Yaskawa INFORM job: miniTRJ0.JBI

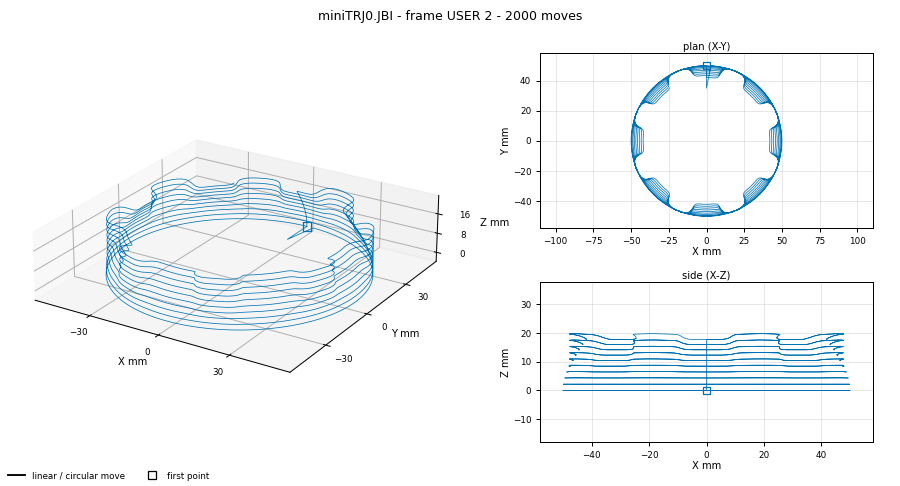
[picture p0: tool path of miniTRJ0.JBI in frame USER 2, 2000 of 2000 moves have a stored position in this frame; points joined in program order, loops and branches not executed]
/JOB
//NAME miniTRJ0
//POS
///NPOS 2000,0,0,0,0,0
///USER 2
///TOOL 1
///POSTYPE USER
///RECTAN
///RCONF 1,0,0,0,0,0,0,0,0,0,0,0,0,0,0,0,0,0,0,0,0,0,0,0
C00000=0.000,50.000,0.000,143.3809,0.0008,0.0000
C00001=0.000,35.000,0.000,143.3809,0.0008,0.0000
C00002=2.896,49.916,0.000,143.4142,-2.1763,0.0000
C00003=5.494,49.697,0.000,143.4861,-2.5054,0.0000
C00004=7.782,49.391,0.000,143.6143,-1.9514,0.0000
C00005=9.349,49.118,0.000,143.7421,-1.4817,0.0000
C00006=10.427,48.901,0.000,143.8463,-1.1243,0.0000
C00007=11.297,48.707,0.000,143.9396,-0.8206,0.0000
C00008=12.176,48.495,0.000,144.0418,-0.5020,0.0000
C00009=13.275,48.206,0.000,144.1803,-0.0901,0.0000
C00010=14.624,47.814,0.000,144.3651,0.4321,0.0000
C00011=16.047,47.355,0.000,144.5758,0.9982,0.0000
C00012=17.369,46.886,0.000,144.7843,1.5341,0.0000
C00013=18.561,46.427,0.000,144.9812,2.0219,0.0000
C00014=19.705,45.953,0.000,155.0622,-25.4971,0.0000
C00015=20.871,45.435,0.000,154.5493,-25.2482,0.0000
C00016=22.138,44.832,0.000,153.9948,-24.9681,0.0000
C00017=23.469,44.150,0.000,153.4198,-24.6638,0.0000
C00018=24.700,43.473,0.000,152.9002,-24.3753,0.0000
C00019=25.682,42.901,0.000,152.4981,-24.1419,0.0000
C00020=26.453,42.429,0.000,152.1923,-23.9575,0.0000
C00021=27.205,41.951,0.000,151.9052,-23.7787,0.0000
C00022=28.121,41.343,0.000,151.5731,-23.5641,0.0000
C00023=29.422,40.427,0.000,151.1462,-23.2751,0.0000
C00024=31.256,39.026,0.000,150.6643,-22.9190,0.0000
C00025=33.248,37.344,0.000,150.8238,-23.2222,0.0000
C00026=35.355,35.355,0.000,152.2782,-24.9479,0.0000
C00027=37.344,33.248,0.000,153.8299,-26.6153,0.0000
C00028=39.026,31.256,0.000,154.1264,-26.8237,0.0000
C00029=40.427,29.422,0.000,153.8428,-26.3144,0.0000
C00030=41.343,28.121,0.000,153.6210,-25.8703,0.0000
C00031=41.951,27.205,0.000,153.4595,-25.5278,0.0000
C00032=42.429,26.453,0.000,153.3270,-25.2337,0.0000
C00033=42.901,25.682,0.000,153.1924,-24.9221,0.0000
C00034=43.473,24.700,0.000,153.0248,-24.5152,0.0000
C00035=44.150,23.469,0.000,152.8218,-23.9932,0.0000
C00036=44.832,22.138,0.000,152.6122,-23.4205,0.0000
C00037=45.435,20.871,0.000,152.4232,-22.8724,0.0000
C00038=45.953,19.705,0.000,152.2582,-22.3690,0.0000
C00039=46.427,18.561,0.000,-177.5317,-34.9939,0.0000
C00040=46.886,17.369,0.000,-178.1225,-35.2012,0.0000
C00041=47.355,16.047,0.000,-178.7751,-35.4180,0.0000
C00042=47.814,14.624,0.000,-179.4684,-35.6337,0.0000
C00043=48.206,13.275,0.000,179.8889,-35.8197,0.0000
C00044=48.495,12.176,0.000,179.3798,-35.9566,0.0000
C00045=48.707,11.297,0.000,178.9849,-36.0561,0.0000
C00046=48.901,10.427,0.000,178.6076,-36.1456,0.0000
C00047=49.118,9.349,0.000,178.1627,-36.2439,0.0000
C00048=49.391,7.782,0.000,177.5765,-36.3612,0.0000
C00049=49.697,5.494,0.000,176.8838,-36.4734,0.0000
C00050=49.916,2.896,0.000,177.2904,-36.5551,0.0000
C00051=50.000,0.000,0.000,-179.9990,-36.6191,0.0000
C00052=49.916,-2.896,0.000,-177.2909,-36.5552,0.0000
C00053=49.697,-5.494,0.000,-176.8841,-36.4733,0.0000
C00054=49.391,-7.782,0.000,-177.5773,-36.3612,0.0000
C00055=49.118,-9.349,0.000,-178.1633,-36.2439,0.0000
C00056=48.901,-10.427,0.000,-178.6081,-36.1456,0.0000
C00057=48.707,-11.297,0.000,-178.9853,-36.0561,0.0000
C00058=48.495,-12.176,0.000,-179.3801,-35.9565,0.0000
C00059=48.206,-13.275,0.000,-179.8890,-35.8196,0.0000
C00060=47.814,-14.624,0.000,179.4684,-35.6336,0.0000
C00061=47.355,-16.047,0.000,178.7752,-35.4179,0.0000
C00062=46.886,-17.369,0.000,178.1227,-35.2010,0.0000
C00063=46.427,-18.561,0.000,177.5319,-34.9937,0.0000
C00064=45.953,-19.705,0.000,-152.2579,-22.3690,0.0000
C00065=45.435,-20.871,0.000,-152.4230,-22.8724,0.0000
C00066=44.832,-22.138,0.000,-152.6120,-23.4205,0.0000
C00067=44.150,-23.469,0.000,-152.8217,-23.9933,0.0000
C00068=43.473,-24.700,0.000,-153.0248,-24.5153,0.0000
C00069=42.901,-25.682,0.000,-153.1925,-24.9223,0.0000
C00070=42.429,-26.453,0.000,-153.3272,-25.2339,0.0000
C00071=41.951,-27.205,0.000,-153.4597,-25.5281,0.0000
C00072=41.343,-28.121,0.000,-153.6213,-25.8707,0.0000
C00073=40.427,-29.422,0.000,-153.8432,-26.3148,0.0000
C00074=39.026,-31.256,0.000,-154.1266,-26.8239,0.0000
C00075=37.344,-33.248,0.000,-153.8302,-26.6155,0.0000
C00076=35.355,-35.355,0.000,-152.2770,-24.9466,0.0000
C00077=33.248,-37.344,0.000,-150.8240,-23.2225,0.0000
C00078=31.256,-39.026,0.000,-150.6645,-22.9191,0.0000
C00079=29.422,-40.427,0.000,-151.1466,-23.2756,0.0000
C00080=28.121,-41.343,0.000,-151.5735,-23.5644,0.0000
C00081=27.205,-41.951,0.000,-151.9055,-23.7790,0.0000
C00082=26.453,-42.429,0.000,-152.1925,-23.9578,0.0000
C00083=25.682,-42.901,0.000,-152.4983,-24.1420,0.0000
C00084=24.700,-43.473,0.000,-152.9003,-24.3754,0.0000
C00085=23.469,-44.150,0.000,-153.4199,-24.6637,0.0000
C00086=22.138,-44.832,0.000,-153.9949,-24.9680,0.0000
C00087=20.871,-45.435,0.000,-154.5494,-25.2480,0.0000
C00088=19.705,-45.953,0.000,-155.0622,-25.4968,0.0000
C00089=18.561,-46.427,0.000,-144.9812,2.0219,0.0000
C00090=17.369,-46.886,0.000,-144.7843,1.5341,0.0000
C00091=16.047,-47.355,0.000,-144.5758,0.9982,0.0000
C00092=14.624,-47.814,0.000,-144.3651,0.4321,0.0000
C00093=13.275,-48.206,0.000,-144.1803,-0.0901,0.0000
C00094=12.176,-48.495,0.000,-144.0418,-0.5020,0.0000
C00095=11.297,-48.707,0.000,-143.9396,-0.8206,0.0000
C00096=10.427,-48.901,0.000,-143.8463,-1.1243,0.0000
C00097=9.349,-49.118,0.000,-143.7421,-1.4817,0.0000
C00098=7.782,-49.391,0.000,-143.6143,-1.9514,0.0000
C00099=5.494,-49.697,0.000,-143.4861,-2.5054,0.0000
C00100=2.896,-49.916,0.000,-143.4142,-2.1763,0.0000
C00101=0.000,-50.000,0.000,-143.3809,0.0008,0.0000
C00102=0.000,-50.000,0.000,-143.3809,0.0008,0.0000
C00103=-2.896,-49.916,0.000,-143.4141,2.1759,0.0000
C00104=-5.494,-49.697,0.000,-143.4861,2.5052,0.0000
C00105=-7.782,-49.391,0.000,-143.6143,1.9508,0.0000
C00106=-9.349,-49.118,0.000,-143.7421,1.4812,0.0000
C00107=-10.427,-48.901,0.000,-143.8463,1.1239,0.0000
C00108=-11.297,-48.707,0.000,-143.9396,0.8203,0.0000
C00109=-12.176,-48.495,0.000,-144.0419,0.5018,0.0000
C00110=-13.275,-48.206,0.000,-144.1804,0.0900,0.0000
C00111=-14.624,-47.814,0.000,-144.3652,-0.4320,0.0000
C00112=-16.047,-47.355,0.000,-144.5759,-0.9981,0.0000
C00113=-17.369,-46.886,0.000,-144.7845,-1.5339,0.0000
C00114=-18.561,-46.427,0.000,-144.9813,-2.0217,0.0000
C00115=-19.705,-45.953,0.000,-155.0622,25.4971,0.0000
C00116=-20.871,-45.435,0.000,-154.5493,25.2482,0.0000
C00117=-22.138,-44.832,0.000,-153.9948,24.9681,0.0000
C00118=-23.469,-44.150,0.000,-153.4198,24.6638,0.0000
C00119=-24.700,-43.473,0.000,-152.9002,24.3753,0.0000
C00120=-25.682,-42.901,0.000,-152.4981,24.1419,0.0000
C00121=-26.453,-42.429,0.000,-152.1923,23.9575,0.0000
C00122=-27.205,-41.951,0.000,-151.9052,23.7787,0.0000
C00123=-28.121,-41.343,0.000,-151.5731,23.5641,0.0000
C00124=-29.422,-40.427,0.000,-151.1462,23.2751,0.0000
C00125=-31.256,-39.026,0.000,-150.6643,22.9190,0.0000
C00126=-33.248,-37.344,0.000,-150.8238,23.2222,0.0000
C00127=-35.355,-35.355,0.000,-152.2782,24.9479,0.0000
C00128=-37.344,-33.248,0.000,-153.8299,26.6153,0.0000
C00129=-39.026,-31.256,0.000,-154.1264,26.8237,0.0000
C00130=-40.427,-29.422,0.000,-153.8428,26.3144,0.0000
C00131=-41.343,-28.121,0.000,-153.6210,25.8703,0.0000
C00132=-41.951,-27.205,0.000,-153.4595,25.5278,0.0000
C00133=-42.429,-26.453,0.000,-153.3270,25.2337,0.0000
C00134=-42.901,-25.682,0.000,-153.1924,24.9221,0.0000
C00135=-43.473,-24.700,0.000,-153.0248,24.5152,0.0000
C00136=-44.150,-23.469,0.000,-152.8218,23.9932,0.0000
C00137=-44.832,-22.138,0.000,-152.6122,23.4205,0.0000
C00138=-45.435,-20.871,0.000,-152.4232,22.8724,0.0000
C00139=-45.953,-19.705,0.000,-152.2582,22.3690,0.0000
C00140=-46.427,-18.561,0.000,177.5317,34.9939,0.0000
C00141=-46.886,-17.369,0.000,178.1225,35.2012,0.0000
C00142=-47.355,-16.047,0.000,178.7751,35.4180,0.0000
C00143=-47.814,-14.624,0.000,179.4684,35.6337,0.0000
C00144=-48.206,-13.275,0.000,-179.8889,35.8197,0.0000
C00145=-48.495,-12.176,0.000,-179.3798,35.9566,0.0000
C00146=-48.707,-11.297,0.000,-178.9849,36.0561,0.0000
C00147=-48.901,-10.427,0.000,-178.6076,36.1456,0.0000
C00148=-49.118,-9.349,0.000,-178.1627,36.2439,0.0000
C00149=-49.391,-7.782,0.000,-177.5765,36.3612,0.0000
C00150=-49.697,-5.494,0.000,-176.8838,36.4734,0.0000
C00151=-49.916,-2.896,0.000,-177.2904,36.5551,0.0000
C00152=-50.000,0.000,0.000,179.9990,36.6191,0.0000
C00153=-49.916,2.896,0.000,177.2909,36.5552,0.0000
C00154=-49.697,5.494,0.000,176.8841,36.4733,0.0000
C00155=-49.391,7.782,0.000,177.5773,36.3612,0.0000
C00156=-49.118,9.349,0.000,178.1633,36.2439,0.0000
C00157=-48.901,10.427,0.000,178.6081,36.1456,0.0000
C00158=-48.707,11.297,0.000,178.9853,36.0561,0.0000
C00159=-48.495,12.176,0.000,179.3801,35.9565,0.0000
C00160=-48.206,13.275,0.000,179.8890,35.8196,0.0000
C00161=-47.814,14.624,0.000,-179.4684,35.6336,0.0000
C00162=-47.355,16.047,0.000,-178.7752,35.4179,0.0000
C00163=-46.886,17.369,0.000,-178.1227,35.2010,0.0000
C00164=-46.427,18.561,0.000,-177.5319,34.9937,0.0000
C00165=-45.953,19.705,0.000,152.2579,22.3690,0.0000
C00166=-45.435,20.871,0.000,152.4230,22.8724,0.0000
C00167=-44.832,22.138,0.000,152.6120,23.4205,0.0000
C00168=-44.150,23.469,0.000,152.8217,23.9933,0.0000
C00169=-43.473,24.700,0.000,153.0248,24.5153,0.0000
C00170=-42.901,25.682,0.000,153.1925,24.9223,0.0000
C00171=-42.429,26.453,0.000,153.3272,25.2339,0.0000
C00172=-41.951,27.205,0.000,153.4597,25.5281,0.0000
C00173=-41.343,28.121,0.000,153.6213,25.8707,0.0000
C00174=-40.427,29.422,0.000,153.8432,26.3148,0.0000
C00175=-39.026,31.256,0.000,154.1266,26.8239,0.0000
C00176=-37.344,33.248,0.000,153.8302,26.6155,0.0000
C00177=-35.355,35.355,0.000,152.2770,24.9466,0.0000
C00178=-33.248,37.344,0.000,150.8240,23.2225,0.0000
C00179=-31.256,39.026,0.000,150.6645,22.9191,0.0000
C00180=-29.422,40.427,0.000,151.1466,23.2756,0.0000
C00181=-28.121,41.343,0.000,151.5735,23.5644,0.0000
C00182=-27.205,41.951,0.000,151.9055,23.7790,0.0000
C00183=-26.453,42.429,0.000,152.1925,23.9578,0.0000
C00184=-25.682,42.901,0.000,152.4983,24.1420,0.0000
C00185=-24.700,43.473,0.000,152.9003,24.3754,0.0000
C00186=-23.469,44.150,0.000,153.4199,24.6637,0.0000
C00187=-22.138,44.832,0.000,153.9949,24.9680,0.0000
C00188=-20.871,45.435,0.000,154.5494,25.2480,0.0000
C00189=-19.705,45.953,0.000,155.0622,25.4968,0.0000
C00190=-18.561,46.427,0.000,144.9813,-2.0217,0.0000
C00191=-17.369,46.886,0.000,144.7845,-1.5339,0.0000
C00192=-16.047,47.355,0.000,144.5759,-0.9981,0.0000
C00193=-14.624,47.814,0.000,144.3652,-0.4320,0.0000
C00194=-13.275,48.206,0.000,144.1804,0.0900,0.0000
C00195=-12.176,48.495,0.000,144.0419,0.5018,0.0000
C00196=-11.297,48.707,0.000,143.9396,0.8203,0.0000
C00197=-10.427,48.901,0.000,143.8463,1.1239,0.0000
C00198=-9.349,49.118,0.000,143.7421,1.4812,0.0000
C00199=-7.782,49.391,0.000,143.6143,1.9508,0.0000
C00200=-5.494,49.697,0.000,143.4861,2.5052,0.0000
C00201=-2.896,49.916,0.000,143.4141,2.1759,0.0000
C00202=0.000,50.000,0.000,143.3809,0.0008,0.0000
C00203=0.000,49.846,2.195,142.7871,0.0008,0.0000
C00204=2.882,49.762,2.195,142.8227,-2.2150,0.0000
C00205=5.471,49.545,2.195,142.8908,-2.4632,0.0000
C00206=7.753,49.245,2.195,143.0117,-1.8435,0.0000
C00207=9.315,48.989,2.196,143.1359,-1.3366,0.0000
C00208=10.389,48.795,2.197,143.2401,-0.9560,0.0000
C00209=11.257,48.629,2.198,143.3352,-0.6346,0.0000
C00210=12.134,48.445,2.199,143.4401,-0.2988,0.0000
C00211=13.230,48.181,2.199,143.5809,0.1341,0.0000
C00212=14.582,47.809,2.200,143.7697,0.6839,0.0000
C00213=16.014,47.361,2.200,143.9865,1.2808,0.0000
C00214=17.348,46.893,2.200,144.2028,1.8461,0.0000
C00215=18.554,46.430,2.200,144.4088,2.3605,0.0000
C00216=19.712,45.950,2.200,154.8156,-26.1236,0.0000
C00217=20.891,45.426,2.200,154.2738,-25.8594,0.0000
C00218=22.166,44.813,2.200,153.6898,-25.5604,0.0000
C00219=23.495,44.117,2.200,153.0860,-25.2351,0.0000
C00220=24.714,43.424,2.199,152.5422,-24.9264,0.0000
C00221=25.676,42.836,2.199,152.1226,-24.6771,0.0000
C00222=26.426,42.346,2.198,151.8021,-24.4802,0.0000
C00223=27.157,41.850,2.197,151.5007,-24.2879,0.0000
C00224=28.054,41.227,2.196,151.1523,-24.0540,0.0000
C00225=29.339,40.304,2.195,150.7028,-23.7323,0.0000
C00226=31.165,38.902,2.195,150.1829,-23.3183,0.0000
C00227=33.149,37.225,2.195,150.2905,-23.5560,0.0000
C00228=35.246,35.246,2.195,151.7659,-25.3187,0.0000
C00229=37.225,33.149,2.195,153.3450,-27.0199,0.0000
C00230=38.902,31.165,2.195,153.5809,-27.1689,0.0000
C00231=40.304,29.339,2.195,153.2459,-26.6124,0.0000
C00232=41.227,28.054,2.196,152.9964,-26.1408,0.0000
C00233=41.850,27.157,2.197,152.8199,-25.7796,0.0000
C00234=42.346,26.426,2.198,152.6780,-25.4699,0.0000
C00235=42.836,25.676,2.199,152.5351,-25.1428,0.0000
C00236=43.424,24.714,2.199,152.3569,-24.7173,0.0000
C00237=44.117,23.495,2.200,152.1408,-24.1705,0.0000
C00238=44.813,22.166,2.200,151.9184,-23.5689,0.0000
C00239=45.426,20.891,2.200,151.7187,-22.9922,0.0000
C00240=45.950,19.712,2.200,151.5461,-22.4615,0.0000
C00241=46.430,18.554,2.200,-177.0981,-35.5564,0.0000
C00242=46.893,17.348,2.200,-177.7244,-35.7758,0.0000
C00243=47.361,16.014,2.200,-178.4168,-36.0031,0.0000
C00244=47.809,14.582,2.200,-179.1522,-36.2274,0.0000
C00245=48.181,13.230,2.199,-179.8333,-36.4190,0.0000
C00246=48.445,12.134,2.199,179.6280,-36.5594,0.0000
C00247=48.629,11.257,2.198,179.2089,-36.6622,0.0000
C00248=48.795,10.389,2.197,178.8068,-36.7540,0.0000
C00249=48.989,9.315,2.196,178.3295,-36.8524,0.0000
C00250=49.245,7.753,2.195,177.6925,-36.9660,0.0000
C00251=49.545,5.471,2.195,176.9123,-37.0692,0.0000
C00252=49.762,2.882,2.195,177.2208,-37.1449,0.0000
C00253=49.846,0.000,2.195,-179.9990,-37.2129,0.0000
C00254=49.762,-2.882,2.195,-177.2212,-37.1450,0.0000
C00255=49.545,-5.471,2.195,-176.9127,-37.0691,0.0000
C00256=49.245,-7.753,2.195,-177.6932,-36.9659,0.0000
C00257=48.989,-9.315,2.196,-178.3302,-36.8524,0.0000
C00258=48.795,-10.389,2.197,-178.8073,-36.7540,0.0000
C00259=48.629,-11.257,2.198,-179.2093,-36.6621,0.0000
C00260=48.445,-12.134,2.199,-179.6283,-36.5593,0.0000
C00261=48.181,-13.230,2.199,179.8332,-36.4189,0.0000
C00262=47.809,-14.582,2.200,179.1522,-36.2273,0.0000
C00263=47.361,-16.014,2.200,178.4168,-36.0030,0.0000
C00264=46.893,-17.348,2.200,177.7245,-35.7757,0.0000
C00265=46.430,-18.554,2.200,177.0983,-35.5563,0.0000
C00266=45.950,-19.712,2.200,-151.5459,-22.4615,0.0000
C00267=45.426,-20.891,2.200,-151.7185,-22.9922,0.0000
C00268=44.813,-22.166,2.200,-151.9182,-23.5690,0.0000
C00269=44.117,-23.495,2.200,-152.1407,-24.1705,0.0000
C00270=43.424,-24.714,2.199,-152.3570,-24.7174,0.0000
C00271=42.836,-25.676,2.199,-152.5352,-25.1430,0.0000
C00272=42.346,-26.426,2.198,-152.6781,-25.4702,0.0000
C00273=41.850,-27.157,2.197,-152.8202,-25.7800,0.0000
C00274=41.227,-28.054,2.196,-152.9968,-26.1412,0.0000
C00275=40.304,-29.339,2.195,-153.2463,-26.6128,0.0000
C00276=38.902,-31.165,2.195,-153.5811,-27.1692,0.0000
C00277=37.225,-33.149,2.195,-153.3453,-27.0201,0.0000
C00278=35.246,-35.246,2.195,-151.7648,-25.3174,0.0000
C00279=33.149,-37.225,2.195,-150.2907,-23.5563,0.0000
C00280=31.165,-38.902,2.195,-150.1831,-23.3185,0.0000
C00281=29.339,-40.304,2.195,-150.7032,-23.7328,0.0000
C00282=28.054,-41.227,2.196,-151.1526,-24.0544,0.0000
C00283=27.157,-41.850,2.197,-151.5010,-24.2882,0.0000
C00284=26.426,-42.346,2.198,-151.8023,-24.4804,0.0000
C00285=25.676,-42.836,2.199,-152.1228,-24.6773,0.0000
C00286=24.714,-43.424,2.199,-152.5424,-24.9265,0.0000
C00287=23.495,-44.117,2.200,-153.0861,-25.2350,0.0000
C00288=22.166,-44.813,2.200,-153.6898,-25.5603,0.0000
C00289=20.891,-45.426,2.200,-154.2738,-25.8592,0.0000
C00290=19.712,-45.950,2.200,-154.8157,-26.1234,0.0000
C00291=18.554,-46.430,2.200,-144.4088,2.3605,0.0000
C00292=17.348,-46.893,2.200,-144.2028,1.8461,0.0000
C00293=16.014,-47.361,2.200,-143.9865,1.2808,0.0000
C00294=14.582,-47.809,2.200,-143.7697,0.6839,0.0000
C00295=13.230,-48.181,2.199,-143.5809,0.1341,0.0000
C00296=12.134,-48.445,2.199,-143.4401,-0.2988,0.0000
C00297=11.257,-48.629,2.198,-143.3352,-0.6346,0.0000
C00298=10.389,-48.795,2.197,-143.2401,-0.9560,0.0000
C00299=9.315,-48.989,2.196,-143.1359,-1.3366,0.0000
C00300=7.753,-49.245,2.195,-143.0117,-1.8435,0.0000
C00301=5.471,-49.545,2.195,-142.8908,-2.4632,0.0000
C00302=2.882,-49.762,2.195,-142.8227,-2.2150,0.0000
C00303=0.000,-49.846,2.195,-142.7871,0.0008,0.0000
C00304=0.000,-49.846,2.195,-142.7871,0.0008,0.0000
C00305=-2.882,-49.762,2.195,-142.8226,2.2147,0.0000
C00306=-5.471,-49.545,2.195,-142.8908,2.4630,0.0000
C00307=-7.753,-49.245,2.195,-143.0117,1.8429,0.0000
C00308=-9.315,-48.989,2.196,-143.1359,1.3361,0.0000
C00309=-10.389,-48.795,2.197,-143.2401,0.9556,0.0000
C00310=-11.257,-48.629,2.198,-143.3353,0.6342,0.0000
C00311=-12.134,-48.445,2.199,-143.4401,0.2985,0.0000
C00312=-13.230,-48.181,2.199,-143.5810,-0.1342,0.0000
C00313=-14.582,-47.809,2.200,-143.7698,-0.6839,0.0000
C00314=-16.014,-47.361,2.200,-143.9866,-1.2807,0.0000
C00315=-17.348,-46.893,2.200,-144.2029,-1.8459,0.0000
C00316=-18.554,-46.430,2.200,-144.4089,-2.3603,0.0000
C00317=-19.712,-45.950,2.200,-154.8156,26.1236,0.0000
C00318=-20.891,-45.426,2.200,-154.2738,25.8594,0.0000
C00319=-22.166,-44.813,2.200,-153.6898,25.5604,0.0000
C00320=-23.495,-44.117,2.200,-153.0860,25.2351,0.0000
C00321=-24.714,-43.424,2.199,-152.5422,24.9264,0.0000
C00322=-25.676,-42.836,2.199,-152.1226,24.6771,0.0000
C00323=-26.426,-42.346,2.198,-151.8021,24.4802,0.0000
C00324=-27.157,-41.850,2.197,-151.5007,24.2879,0.0000
C00325=-28.054,-41.227,2.196,-151.1523,24.0540,0.0000
C00326=-29.339,-40.304,2.195,-150.7028,23.7323,0.0000
C00327=-31.165,-38.902,2.195,-150.1829,23.3183,0.0000
C00328=-33.149,-37.225,2.195,-150.2905,23.5560,0.0000
C00329=-35.246,-35.246,2.195,-151.7659,25.3187,0.0000
C00330=-37.225,-33.149,2.195,-153.3450,27.0199,0.0000
C00331=-38.902,-31.165,2.195,-153.5809,27.1689,0.0000
C00332=-40.304,-29.339,2.195,-153.2459,26.6124,0.0000
C00333=-41.227,-28.054,2.196,-152.9964,26.1408,0.0000
C00334=-41.850,-27.157,2.197,-152.8199,25.7796,0.0000
C00335=-42.346,-26.426,2.198,-152.6780,25.4699,0.0000
C00336=-42.836,-25.676,2.199,-152.5351,25.1428,0.0000
C00337=-43.424,-24.714,2.199,-152.3569,24.7173,0.0000
C00338=-44.117,-23.495,2.200,-152.1408,24.1705,0.0000
C00339=-44.813,-22.166,2.200,-151.9184,23.5689,0.0000
C00340=-45.426,-20.891,2.200,-151.7187,22.9922,0.0000
C00341=-45.950,-19.712,2.200,-151.5461,22.4615,0.0000
C00342=-46.430,-18.554,2.200,177.0981,35.5564,0.0000
C00343=-46.893,-17.348,2.200,177.7244,35.7758,0.0000
C00344=-47.361,-16.014,2.200,178.4168,36.0031,0.0000
C00345=-47.809,-14.582,2.200,179.1522,36.2274,0.0000
C00346=-48.181,-13.230,2.199,179.8333,36.4190,0.0000
C00347=-48.445,-12.134,2.199,-179.6280,36.5594,0.0000
C00348=-48.629,-11.257,2.198,-179.2089,36.6622,0.0000
C00349=-48.795,-10.389,2.197,-178.8068,36.7540,0.0000
C00350=-48.989,-9.315,2.196,-178.3295,36.8524,0.0000
C00351=-49.245,-7.753,2.195,-177.6925,36.9660,0.0000
C00352=-49.545,-5.471,2.195,-176.9123,37.0692,0.0000
C00353=-49.762,-2.882,2.195,-177.2208,37.1449,0.0000
C00354=-49.846,0.000,2.195,179.9990,37.2129,0.0000
C00355=-49.762,2.882,2.195,177.2212,37.1450,0.0000
C00356=-49.545,5.471,2.195,176.9127,37.0691,0.0000
C00357=-49.245,7.753,2.195,177.6932,36.9659,0.0000
C00358=-48.989,9.315,2.196,178.3302,36.8524,0.0000
C00359=-48.795,10.389,2.197,178.8073,36.7540,0.0000
C00360=-48.629,11.257,2.198,179.2093,36.6621,0.0000
C00361=-48.445,12.134,2.199,179.6283,36.5593,0.0000
C00362=-48.181,13.230,2.199,-179.8332,36.4189,0.0000
C00363=-47.809,14.582,2.200,-179.1522,36.2273,0.0000
C00364=-47.361,16.014,2.200,-178.4168,36.0030,0.0000
C00365=-46.893,17.348,2.200,-177.7245,35.7757,0.0000
C00366=-46.430,18.554,2.200,-177.0983,35.5563,0.0000
C00367=-45.950,19.712,2.200,151.5459,22.4615,0.0000
C00368=-45.426,20.891,2.200,151.7185,22.9922,0.0000
C00369=-44.813,22.166,2.200,151.9182,23.5690,0.0000
C00370=-44.117,23.495,2.200,152.1407,24.1705,0.0000
C00371=-43.424,24.714,2.199,152.3570,24.7174,0.0000
C00372=-42.836,25.676,2.199,152.5352,25.1430,0.0000
C00373=-42.346,26.426,2.198,152.6781,25.4702,0.0000
C00374=-41.850,27.157,2.197,152.8202,25.7800,0.0000
C00375=-41.227,28.054,2.196,152.9968,26.1412,0.0000
C00376=-40.304,29.339,2.195,153.2463,26.6128,0.0000
C00377=-38.902,31.165,2.195,153.5811,27.1692,0.0000
C00378=-37.225,33.149,2.195,153.3453,27.0201,0.0000
C00379=-35.246,35.246,2.195,151.7648,25.3174,0.0000
C00380=-33.149,37.225,2.195,150.2907,23.5563,0.0000
C00381=-31.165,38.902,2.195,150.1831,23.3185,0.0000
C00382=-29.339,40.304,2.195,150.7032,23.7328,0.0000
C00383=-28.054,41.227,2.196,151.1526,24.0544,0.0000
C00384=-27.157,41.850,2.197,151.5010,24.2882,0.0000
C00385=-26.426,42.346,2.198,151.8023,24.4804,0.0000
C00386=-25.676,42.836,2.199,152.1228,24.6773,0.0000
C00387=-24.714,43.424,2.199,152.5424,24.9265,0.0000
C00388=-23.495,44.117,2.200,153.0861,25.2350,0.0000
C00389=-22.166,44.813,2.200,153.6898,25.5603,0.0000
C00390=-20.891,45.426,2.200,154.2738,25.8592,0.0000
C00391=-19.712,45.950,2.200,154.8157,26.1234,0.0000
C00392=-18.554,46.430,2.200,144.4089,-2.3603,0.0000
C00393=-17.348,46.893,2.200,144.2029,-1.8459,0.0000
C00394=-16.014,47.361,2.200,143.9866,-1.2807,0.0000
C00395=-14.582,47.809,2.200,143.7698,-0.6839,0.0000
C00396=-13.230,48.181,2.199,143.5810,-0.1342,0.0000
C00397=-12.134,48.445,2.199,143.4401,0.2985,0.0000
C00398=-11.257,48.629,2.198,143.3353,0.6342,0.0000
C00399=-10.389,48.795,2.197,143.2401,0.9556,0.0000
C00400=-9.315,48.989,2.196,143.1359,1.3361,0.0000
C00401=-7.753,49.245,2.195,143.0117,1.8429,0.0000
C00402=-5.471,49.545,2.195,142.8908,2.4630,0.0000
C00403=-2.882,49.762,2.195,142.8226,2.2147,0.0000
C00404=0.000,49.846,2.195,142.7871,0.0008,0.0000
C00405=0.000,49.410,4.351,142.2720,0.0007,0.0000
C00406=2.842,49.327,4.351,142.3092,-2.2444,0.0000
C00407=5.404,49.114,4.351,142.3736,-2.4180,0.0000
C00408=7.672,48.833,4.355,142.4892,-1.7397,0.0000
C00409=9.218,48.623,4.363,142.6124,-1.2036,0.0000
C00410=10.282,48.495,4.374,142.7197,-0.8069,0.0000
C00411=11.143,48.407,4.384,142.8211,-0.4739,0.0000
C00412=12.014,48.303,4.391,142.9335,-0.1276,0.0000
C00413=13.101,48.111,4.395,143.0816,0.3184,0.0000
C00414=14.461,47.794,4.396,143.2802,0.8931,0.0000
C00415=15.918,47.378,4.398,143.5102,1.5238,0.0000
C00416=17.289,46.913,4.399,143.7405,2.1264,0.0000
C00417=18.533,46.438,4.400,143.9621,2.6774,0.0000
C00418=19.732,45.942,4.400,154.6593,-26.6527,0.0000
C00419=20.948,45.397,4.399,154.0760,-26.3698,0.0000
C00420=22.246,44.758,4.398,153.4514,-26.0501,0.0000
C00421=23.570,44.021,4.396,152.8110,-25.7058,0.0000
C00422=24.756,43.284,4.395,152.2399,-25.3828,0.0000
C00423=25.660,42.651,4.391,151.8041,-25.1271,0.0000
C00424=26.350,42.108,4.384,151.4691,-24.9258,0.0000
C00425=27.021,41.562,4.374,151.1539,-24.7276,0.0000
C00426=27.864,40.900,4.363,150.7913,-24.4822,0.0000
C00427=29.106,39.955,4.355,150.3226,-24.1357,0.0000
C00428=30.908,38.550,4.351,149.7679,-23.6707,0.0000
C00429=32.870,36.889,4.351,149.8283,-23.8474,0.0000
C00430=34.938,34.938,4.351,151.3189,-25.6389,0.0000
C00431=36.889,32.870,4.351,152.9185,-27.3666,0.0000
C00432=38.550,30.908,4.351,153.0982,-27.4607,0.0000
C00433=39.955,29.106,4.355,152.7186,-26.8609,0.0000
C00434=40.900,27.864,4.363,152.4494,-26.3664,0.0000
C00435=41.562,27.021,4.374,152.2657,-25.9900,0.0000
C00436=42.108,26.350,4.384,152.1223,-25.6669,0.0000
C00437=42.651,25.660,4.391,151.9798,-25.3262,0.0000
C00438=43.284,24.756,4.395,151.8006,-24.8854,0.0000
C00439=44.021,23.570,4.396,151.5781,-24.3120,0.0000
C00440=44.758,22.246,4.398,151.3465,-23.6751,0.0000
C00441=45.397,20.948,4.399,151.1361,-23.0596,0.0000
C00442=45.942,19.732,4.400,150.9546,-22.4900,0.0000
C00443=46.438,18.533,4.400,-176.6903,-35.9924,0.0000
C00444=46.913,17.289,4.399,-177.3636,-36.2306,0.0000
C00445=47.378,15.918,4.398,-178.1049,-36.4748,0.0000
C00446=47.794,14.461,4.396,-178.8858,-36.7146,0.0000
C00447=48.111,13.101,4.395,-179.6018,-36.9177,0.0000
C00448=48.303,12.014,4.391,179.8401,-37.0664,0.0000
C00449=48.407,11.143,4.384,179.4052,-37.1774,0.0000
C00450=48.495,10.282,4.374,178.9860,-37.2759,0.0000
C00451=48.623,9.218,4.363,178.4853,-37.3780,0.0000
C00452=48.833,7.672,4.355,177.8073,-37.4905,0.0000
C00453=49.114,5.404,4.351,176.9481,-37.5871,0.0000
C00454=49.327,2.842,4.351,177.1646,-37.6569,0.0000
C00455=49.410,0.000,4.351,-179.9991,-37.7280,0.0000
C00456=49.327,-2.842,4.351,-177.1650,-37.6569,0.0000
C00457=49.114,-5.404,4.351,-176.9485,-37.5870,0.0000
C00458=48.833,-7.672,4.355,-177.8080,-37.4905,0.0000
C00459=48.623,-9.218,4.363,-178.4859,-37.3779,0.0000
C00460=48.495,-10.282,4.374,-178.9865,-37.2759,0.0000
C00461=48.407,-11.143,4.384,-179.4056,-37.1773,0.0000
C00462=48.303,-12.014,4.391,-179.8405,-37.0663,0.0000
C00463=48.111,-13.101,4.395,179.6016,-36.9176,0.0000
C00464=47.794,-14.461,4.396,178.8858,-36.7145,0.0000
C00465=47.378,-15.918,4.398,178.1050,-36.4747,0.0000
C00466=46.913,-17.289,4.399,177.3637,-36.2305,0.0000
C00467=46.438,-18.533,4.400,176.6904,-35.9923,0.0000
C00468=45.942,-19.732,4.400,-150.9544,-22.4899,0.0000
C00469=45.397,-20.948,4.399,-151.1359,-23.0596,0.0000
C00470=44.758,-22.246,4.398,-151.3464,-23.6751,0.0000
C00471=44.021,-23.570,4.396,-151.5781,-24.3121,0.0000
C00472=43.284,-24.756,4.395,-151.8007,-24.8855,0.0000
C00473=42.651,-25.660,4.391,-151.9800,-25.3265,0.0000
C00474=42.108,-26.350,4.384,-152.1225,-25.6672,0.0000
C00475=41.562,-27.021,4.374,-152.2659,-25.9903,0.0000
C00476=40.900,-27.864,4.363,-152.4497,-26.3668,0.0000
C00477=39.955,-29.106,4.355,-152.7190,-26.8614,0.0000
C00478=38.550,-30.908,4.351,-153.0984,-27.4609,0.0000
C00479=36.889,-32.870,4.351,-152.9188,-27.3668,0.0000
C00480=34.938,-34.938,4.351,-151.3179,-25.6377,0.0000
C00481=32.870,-36.889,4.351,-149.8284,-23.8476,0.0000
C00482=30.908,-38.550,4.351,-149.7681,-23.6709,0.0000
C00483=29.106,-39.955,4.355,-150.3230,-24.1362,0.0000
C00484=27.864,-40.900,4.363,-150.7917,-24.4825,0.0000
C00485=27.021,-41.562,4.374,-151.1543,-24.7279,0.0000
C00486=26.350,-42.108,4.384,-151.4694,-24.9261,0.0000
C00487=25.660,-42.651,4.391,-151.8043,-25.1272,0.0000
C00488=24.756,-43.284,4.395,-152.2401,-25.3829,0.0000
C00489=23.570,-44.021,4.396,-152.8111,-25.7058,0.0000
C00490=22.246,-44.758,4.398,-153.4515,-26.0500,0.0000
C00491=20.948,-45.397,4.399,-154.0760,-26.3696,0.0000
C00492=19.732,-45.942,4.400,-154.6593,-26.6525,0.0000
C00493=18.533,-46.438,4.400,-143.9621,2.6774,0.0000
C00494=17.289,-46.913,4.399,-143.7405,2.1264,0.0000
C00495=15.918,-47.378,4.398,-143.5102,1.5238,0.0000
C00496=14.461,-47.794,4.396,-143.2802,0.8931,0.0000
C00497=13.101,-48.111,4.395,-143.0816,0.3184,0.0000
C00498=12.014,-48.303,4.391,-142.9335,-0.1276,0.0000
C00499=11.143,-48.407,4.384,-142.8211,-0.4739,0.0000
C00500=10.282,-48.495,4.374,-142.7197,-0.8069,0.0000
C00501=9.218,-48.623,4.363,-142.6124,-1.2036,0.0000
C00502=7.672,-48.833,4.355,-142.4892,-1.7397,0.0000
C00503=5.404,-49.114,4.351,-142.3736,-2.4180,0.0000
C00504=2.842,-49.327,4.351,-142.3092,-2.2444,0.0000
C00505=0.000,-49.410,4.351,-142.2720,0.0007,0.0000
C00506=0.000,-49.410,4.351,-142.2720,0.0007,0.0000
C00507=-2.842,-49.327,4.351,-142.3091,2.2441,0.0000
C00508=-5.404,-49.114,4.351,-142.3737,2.4177,0.0000
C00509=-7.672,-48.833,4.355,-142.4893,1.7391,0.0000
C00510=-9.218,-48.623,4.363,-142.6124,1.2031,0.0000
C00511=-10.282,-48.495,4.374,-142.7198,0.8065,0.0000
C00512=-11.143,-48.407,4.384,-142.8212,0.4736,0.0000
C00513=-12.014,-48.303,4.391,-142.9336,0.1273,0.0000
C00514=-13.101,-48.111,4.395,-143.0817,-0.3185,0.0000
C00515=-14.461,-47.794,4.396,-143.2803,-0.8932,0.0000
C00516=-15.918,-47.378,4.398,-143.5103,-1.5237,0.0000
C00517=-17.289,-46.913,4.399,-143.7406,-2.1263,0.0000
C00518=-18.533,-46.438,4.400,-143.9622,-2.6772,0.0000
C00519=-19.732,-45.942,4.400,-154.6593,26.6527,0.0000
C00520=-20.948,-45.397,4.399,-154.0760,26.3698,0.0000
C00521=-22.246,-44.758,4.398,-153.4514,26.0501,0.0000
C00522=-23.570,-44.021,4.396,-152.8110,25.7058,0.0000
C00523=-24.756,-43.284,4.395,-152.2399,25.3828,0.0000
C00524=-25.660,-42.651,4.391,-151.8041,25.1271,0.0000
C00525=-26.350,-42.108,4.384,-151.4691,24.9258,0.0000
C00526=-27.021,-41.562,4.374,-151.1539,24.7276,0.0000
C00527=-27.864,-40.900,4.363,-150.7913,24.4822,0.0000
C00528=-29.106,-39.955,4.355,-150.3226,24.1357,0.0000
C00529=-30.908,-38.550,4.351,-149.7679,23.6707,0.0000
C00530=-32.870,-36.889,4.351,-149.8283,23.8474,0.0000
C00531=-34.938,-34.938,4.351,-151.3189,25.6389,0.0000
C00532=-36.889,-32.870,4.351,-152.9185,27.3666,0.0000
C00533=-38.550,-30.908,4.351,-153.0982,27.4607,0.0000
C00534=-39.955,-29.106,4.355,-152.7186,26.8609,0.0000
C00535=-40.900,-27.864,4.363,-152.4494,26.3664,0.0000
C00536=-41.562,-27.021,4.374,-152.2657,25.9900,0.0000
C00537=-42.108,-26.350,4.384,-152.1223,25.6669,0.0000
C00538=-42.651,-25.660,4.391,-151.9798,25.3262,0.0000
C00539=-43.284,-24.756,4.395,-151.8006,24.8854,0.0000
C00540=-44.021,-23.570,4.396,-151.5781,24.3120,0.0000
C00541=-44.758,-22.246,4.398,-151.3465,23.6751,0.0000
C00542=-45.397,-20.948,4.399,-151.1361,23.0596,0.0000
C00543=-45.942,-19.732,4.400,-150.9546,22.4900,0.0000
C00544=-46.438,-18.533,4.400,176.6903,35.9924,0.0000
C00545=-46.913,-17.289,4.399,177.3636,36.2306,0.0000
C00546=-47.378,-15.918,4.398,178.1049,36.4748,0.0000
C00547=-47.794,-14.461,4.396,178.8858,36.7146,0.0000
C00548=-48.111,-13.101,4.395,179.6018,36.9177,0.0000
C00549=-48.303,-12.014,4.391,-179.8401,37.0664,0.0000
C00550=-48.407,-11.143,4.384,-179.4052,37.1774,0.0000
C00551=-48.495,-10.282,4.374,-178.9860,37.2759,0.0000
C00552=-48.623,-9.218,4.363,-178.4853,37.3780,0.0000
C00553=-48.833,-7.672,4.355,-177.8073,37.4905,0.0000
C00554=-49.114,-5.404,4.351,-176.9481,37.5871,0.0000
C00555=-49.327,-2.842,4.351,-177.1646,37.6569,0.0000
C00556=-49.410,0.000,4.351,179.9991,37.7280,0.0000
C00557=-49.327,2.842,4.351,177.1650,37.6569,0.0000
C00558=-49.114,5.404,4.351,176.9485,37.5870,0.0000
C00559=-48.833,7.672,4.355,177.8080,37.4905,0.0000
C00560=-48.623,9.218,4.363,178.4859,37.3779,0.0000
C00561=-48.495,10.282,4.374,178.9865,37.2759,0.0000
C00562=-48.407,11.143,4.384,179.4056,37.1773,0.0000
C00563=-48.303,12.014,4.391,179.8405,37.0663,0.0000
C00564=-48.111,13.101,4.395,-179.6016,36.9176,0.0000
C00565=-47.794,14.461,4.396,-178.8858,36.7145,0.0000
C00566=-47.378,15.918,4.398,-178.1050,36.4747,0.0000
C00567=-46.913,17.289,4.399,-177.3637,36.2305,0.0000
C00568=-46.438,18.533,4.400,-176.6904,35.9923,0.0000
C00569=-45.942,19.732,4.400,150.9544,22.4899,0.0000
C00570=-45.397,20.948,4.399,151.1359,23.0596,0.0000
C00571=-44.758,22.246,4.398,151.3464,23.6751,0.0000
C00572=-44.021,23.570,4.396,151.5781,24.3121,0.0000
C00573=-43.284,24.756,4.395,151.8007,24.8855,0.0000
C00574=-42.651,25.660,4.391,151.9800,25.3265,0.0000
C00575=-42.108,26.350,4.384,152.1225,25.6672,0.0000
C00576=-41.562,27.021,4.374,152.2659,25.9903,0.0000
C00577=-40.900,27.864,4.363,152.4497,26.3668,0.0000
C00578=-39.955,29.106,4.355,152.7190,26.8614,0.0000
C00579=-38.550,30.908,4.351,153.0984,27.4609,0.0000
C00580=-36.889,32.870,4.351,152.9188,27.3668,0.0000
C00581=-34.938,34.938,4.351,151.3179,25.6377,0.0000
C00582=-32.870,36.889,4.351,149.8284,23.8476,0.0000
C00583=-30.908,38.550,4.351,149.7681,23.6709,0.0000
C00584=-29.106,39.955,4.355,150.3230,24.1362,0.0000
C00585=-27.864,40.900,4.363,150.7917,24.4825,0.0000
C00586=-27.021,41.562,4.374,151.1543,24.7279,0.0000
C00587=-26.350,42.108,4.384,151.4694,24.9261,0.0000
C00588=-25.660,42.651,4.391,151.8043,25.1272,0.0000
C00589=-24.756,43.284,4.395,152.2401,25.3829,0.0000
C00590=-23.570,44.021,4.396,152.8111,25.7058,0.0000
C00591=-22.246,44.758,4.398,153.4515,26.0500,0.0000
C00592=-20.948,45.397,4.399,154.0760,26.3696,0.0000
C00593=-19.732,45.942,4.400,154.6593,26.6525,0.0000
C00594=-18.533,46.438,4.400,143.9622,-2.6772,0.0000
C00595=-17.289,46.913,4.399,143.7406,-2.1263,0.0000
C00596=-15.918,47.378,4.398,143.5103,-1.5237,0.0000
C00597=-14.461,47.794,4.396,143.2803,-0.8932,0.0000
C00598=-13.101,48.111,4.395,143.0817,-0.3185,0.0000
C00599=-12.014,48.303,4.391,142.9336,0.1273,0.0000
C00600=-11.143,48.407,4.384,142.8212,0.4736,0.0000
C00601=-10.282,48.495,4.374,142.7198,0.8065,0.0000
C00602=-9.218,48.623,4.363,142.6124,1.2031,0.0000
C00603=-7.672,48.833,4.355,142.4893,1.7391,0.0000
C00604=-5.404,49.114,4.351,142.3737,2.4177,0.0000
C00605=-2.842,49.327,4.351,142.3091,2.2441,0.0000
C00606=0.000,49.410,4.351,142.2720,0.0007,0.0000
C00607=0.000,48.740,6.447,141.8391,0.0007,0.0000
C00608=2.781,48.660,6.446,141.8776,-2.2647,0.0000
C00609=5.301,48.453,6.447,141.9384,-2.3722,0.0000
C00610=7.547,48.199,6.458,142.0493,-1.6436,0.0000
C00611=9.067,48.057,6.484,142.1709,-1.0862,0.0000
C00612=10.113,48.028,6.517,142.2804,-0.6798,0.0000
C00613=10.965,48.058,6.549,142.3874,-0.3407,0.0000
C00614=11.826,48.078,6.572,142.5072,0.0108,0.0000
C00615=12.898,48.000,6.582,142.6629,0.4630,0.0000
C00616=14.270,47.771,6.588,142.8733,1.0613,0.0000
C00617=15.768,47.406,6.592,143.1200,1.7302,0.0000
C00618=17.193,46.944,6.597,143.3691,2.3789,0.0000
C00619=18.501,46.450,6.600,143.6119,2.9769,0.0000
C00620=19.763,45.928,6.600,154.5727,-27.1067,0.0000
C00621=21.037,45.352,6.597,153.9353,-26.8007,0.0000
C00622=22.372,44.670,6.592,153.2600,-26.4566,0.0000
C00623=23.689,43.870,6.588,152.5766,-26.0923,0.0000
C00624=24.821,43.061,6.582,151.9778,-25.7575,0.0000
C00625=25.634,42.359,6.572,151.5303,-25.5007,0.0000
C00626=26.229,41.735,6.549,151.1848,-25.2994,0.0000
C00627=26.810,41.112,6.517,150.8600,-25.0991,0.0000
C00628=27.570,40.393,6.484,150.4885,-24.8468,0.0000
C00629=28.746,39.419,6.458,150.0063,-24.4815,0.0000
C00630=30.513,38.009,6.447,149.4219,-23.9723,0.0000
C00631=32.441,36.374,6.446,149.4409,-24.0946,0.0000
C00632=34.464,34.464,6.447,150.9414,-25.9069,0.0000
C00633=36.374,32.441,6.446,152.5550,-27.6537,0.0000
C00634=38.009,30.513,6.447,152.6847,-27.6990,0.0000
C00635=39.419,28.746,6.458,152.2668,-27.0619,0.0000
C00636=40.393,27.570,6.484,151.9826,-26.5510,0.0000
C00637=41.112,26.810,6.517,151.7954,-26.1652,0.0000
C00638=41.735,26.229,6.549,151.6536,-25.8332,0.0000
C00639=42.359,25.634,6.572,151.5152,-25.4835,0.0000
C00640=43.061,24.821,6.582,151.3397,-25.0324,0.0000
C00641=43.870,23.689,6.588,151.1132,-24.4327,0.0000
C00642=44.670,22.372,6.592,150.8723,-23.7546,0.0000
C00643=45.352,21.037,6.597,150.6493,-23.0906,0.0000
C00644=45.928,19.763,6.600,150.4567,-22.4703,0.0000
C00645=46.450,18.501,6.600,-176.3039,-36.3311,0.0000
C00646=46.944,17.193,6.597,-177.0365,-36.5942,0.0000
C00647=47.406,15.768,6.592,-177.8374,-36.8604,0.0000
C00648=47.771,14.270,6.588,-178.6690,-37.1193,0.0000
C00649=48.000,12.898,6.582,-179.4176,-37.3356,0.0000
C00650=48.078,11.826,6.572,-179.9864,-37.4928,0.0000
C00651=48.058,10.965,6.549,179.5699,-37.6118,0.0000
C00652=48.028,10.113,6.517,179.1406,-37.7165,0.0000
C00653=48.057,9.067,6.484,178.6249,-37.8211,0.0000
C00654=48.199,7.547,6.458,177.9160,-37.9323,0.0000
C00655=48.453,5.301,6.447,176.9882,-38.0231,0.0000
C00656=48.660,2.781,6.446,177.1222,-38.0873,0.0000
C00657=48.740,0.000,6.447,-179.9992,-38.1609,0.0000
C00658=48.660,-2.781,6.446,-177.1225,-38.0874,0.0000
C00659=48.453,-5.301,6.447,-176.9886,-38.0231,0.0000
C00660=48.199,-7.547,6.458,-177.9168,-37.9323,0.0000
C00661=48.057,-9.067,6.484,-178.6256,-37.8211,0.0000
C00662=48.028,-10.113,6.517,-179.1411,-37.7164,0.0000
C00663=48.058,-10.965,6.549,-179.5704,-37.6118,0.0000
C00664=48.078,-11.826,6.572,179.9860,-37.4927,0.0000
C00665=48.000,-12.898,6.582,179.4174,-37.3356,0.0000
C00666=47.771,-14.270,6.588,178.6689,-37.1192,0.0000
C00667=47.406,-15.768,6.592,177.8374,-36.8604,0.0000
C00668=46.944,-17.193,6.597,177.0366,-36.5941,0.0000
C00669=46.450,-18.501,6.600,176.3040,-36.3310,0.0000
C00670=45.928,-19.763,6.600,-150.4565,-22.4702,0.0000
C00671=45.352,-21.037,6.597,-150.6491,-23.0906,0.0000
C00672=44.670,-22.372,6.592,-150.8722,-23.7547,0.0000
C00673=43.870,-23.689,6.588,-151.1132,-24.4328,0.0000
C00674=43.061,-24.821,6.582,-151.3398,-25.0326,0.0000
C00675=42.359,-25.634,6.572,-151.5154,-25.4837,0.0000
C00676=41.735,-26.229,6.549,-151.6538,-25.8335,0.0000
C00677=41.112,-26.810,6.517,-151.7957,-26.1655,0.0000
C00678=40.393,-27.570,6.484,-151.9829,-26.5514,0.0000
C00679=39.419,-28.746,6.458,-152.2672,-27.0624,0.0000
C00680=38.009,-30.513,6.447,-152.6849,-27.6993,0.0000
C00681=36.374,-32.441,6.446,-152.5552,-27.6539,0.0000
C00682=34.464,-34.464,6.447,-150.9405,-25.9058,0.0000
C00683=32.441,-36.374,6.446,-149.4410,-24.0949,0.0000
C00684=30.513,-38.009,6.447,-149.4222,-23.9726,0.0000
C00685=28.746,-39.419,6.458,-150.0067,-24.4819,0.0000
C00686=27.570,-40.393,6.484,-150.4889,-24.8471,0.0000
C00687=26.810,-41.112,6.517,-150.8603,-25.0994,0.0000
C00688=26.229,-41.735,6.549,-151.1851,-25.2997,0.0000
C00689=25.634,-42.359,6.572,-151.5305,-25.5009,0.0000
C00690=24.821,-43.061,6.582,-151.9780,-25.7576,0.0000
C00691=23.689,-43.870,6.588,-152.5767,-26.0924,0.0000
C00692=22.372,-44.670,6.592,-153.2600,-26.4565,0.0000
C00693=21.037,-45.352,6.597,-153.9354,-26.8006,0.0000
C00694=19.763,-45.928,6.600,-154.5727,-27.1065,0.0000
C00695=18.501,-46.450,6.600,-143.6119,2.9769,0.0000
C00696=17.193,-46.944,6.597,-143.3691,2.3789,0.0000
C00697=15.768,-47.406,6.592,-143.1200,1.7302,0.0000
C00698=14.270,-47.771,6.588,-142.8733,1.0613,0.0000
C00699=12.898,-48.000,6.582,-142.6629,0.4630,0.0000
C00700=11.826,-48.078,6.572,-142.5072,0.0108,0.0000
C00701=10.965,-48.058,6.549,-142.3874,-0.3407,0.0000
C00702=10.113,-48.028,6.517,-142.2804,-0.6798,0.0000
C00703=9.067,-48.057,6.484,-142.1709,-1.0862,0.0000
C00704=7.547,-48.199,6.458,-142.0493,-1.6436,0.0000
C00705=5.301,-48.453,6.447,-141.9384,-2.3722,0.0000
C00706=2.781,-48.660,6.446,-141.8776,-2.2647,0.0000
C00707=0.000,-48.740,6.447,-141.8391,0.0007,0.0000
C00708=0.000,-48.740,6.447,-141.8391,0.0007,0.0000
C00709=-2.781,-48.660,6.446,-141.8775,2.2645,0.0000
C00710=-5.301,-48.453,6.447,-141.9385,2.3719,0.0000
C00711=-7.547,-48.199,6.458,-142.0494,1.6430,0.0000
C00712=-9.067,-48.057,6.484,-142.1709,1.0857,0.0000
C00713=-10.113,-48.028,6.517,-142.2805,0.6794,0.0000
C00714=-10.965,-48.058,6.549,-142.3874,0.3403,0.0000
C00715=-11.826,-48.078,6.572,-142.5073,-0.0111,0.0000
C00716=-12.898,-48.000,6.582,-142.6630,-0.4632,0.0000
C00717=-14.270,-47.771,6.588,-142.8734,-1.0614,0.0000
C00718=-15.768,-47.406,6.592,-143.1200,-1.7301,0.0000
C00719=-17.193,-46.944,6.597,-143.3692,-2.3789,0.0000
C00720=-18.501,-46.450,6.600,-143.6120,-2.9768,0.0000
C00721=-19.763,-45.928,6.600,-154.5727,27.1067,0.0000
C00722=-21.037,-45.352,6.597,-153.9353,26.8007,0.0000
C00723=-22.372,-44.670,6.592,-153.2600,26.4566,0.0000
C00724=-23.689,-43.870,6.588,-152.5766,26.0923,0.0000
C00725=-24.821,-43.061,6.582,-151.9778,25.7575,0.0000
C00726=-25.634,-42.359,6.572,-151.5303,25.5007,0.0000
C00727=-26.229,-41.735,6.549,-151.1848,25.2994,0.0000
C00728=-26.810,-41.112,6.517,-150.8600,25.0991,0.0000
C00729=-27.570,-40.393,6.484,-150.4885,24.8468,0.0000
C00730=-28.746,-39.419,6.458,-150.0063,24.4815,0.0000
C00731=-30.513,-38.009,6.447,-149.4219,23.9723,0.0000
C00732=-32.441,-36.374,6.446,-149.4409,24.0946,0.0000
C00733=-34.464,-34.464,6.447,-150.9414,25.9069,0.0000
C00734=-36.374,-32.441,6.446,-152.5550,27.6537,0.0000
C00735=-38.009,-30.513,6.447,-152.6847,27.6990,0.0000
C00736=-39.419,-28.746,6.458,-152.2668,27.0619,0.0000
C00737=-40.393,-27.570,6.484,-151.9826,26.5510,0.0000
C00738=-41.112,-26.810,6.517,-151.7954,26.1652,0.0000
C00739=-41.735,-26.229,6.549,-151.6536,25.8332,0.0000
C00740=-42.359,-25.634,6.572,-151.5152,25.4835,0.0000
C00741=-43.061,-24.821,6.582,-151.3397,25.0324,0.0000
C00742=-43.870,-23.689,6.588,-151.1132,24.4327,0.0000
C00743=-44.670,-22.372,6.592,-150.8723,23.7546,0.0000
C00744=-45.352,-21.037,6.597,-150.6493,23.0906,0.0000
C00745=-45.928,-19.763,6.600,-150.4567,22.4703,0.0000
C00746=-46.450,-18.501,6.600,176.3039,36.3311,0.0000
C00747=-46.944,-17.193,6.597,177.0365,36.5942,0.0000
C00748=-47.406,-15.768,6.592,177.8374,36.8604,0.0000
C00749=-47.771,-14.270,6.588,178.6690,37.1193,0.0000
C00750=-48.000,-12.898,6.582,179.4176,37.3356,0.0000
C00751=-48.078,-11.826,6.572,179.9864,37.4928,0.0000
C00752=-48.058,-10.965,6.549,-179.5699,37.6118,0.0000
C00753=-48.028,-10.113,6.517,-179.1406,37.7165,0.0000
C00754=-48.057,-9.067,6.484,-178.6249,37.8211,0.0000
C00755=-48.199,-7.547,6.458,-177.9160,37.9323,0.0000
C00756=-48.453,-5.301,6.447,-176.9882,38.0231,0.0000
C00757=-48.660,-2.781,6.446,-177.1222,38.0873,0.0000
C00758=-48.740,0.000,6.447,179.9992,38.1609,0.0000
C00759=-48.660,2.781,6.446,177.1225,38.0874,0.0000
C00760=-48.453,5.301,6.447,176.9886,38.0231,0.0000
C00761=-48.199,7.547,6.458,177.9168,37.9323,0.0000
C00762=-48.057,9.067,6.484,178.6256,37.8211,0.0000
C00763=-48.028,10.113,6.517,179.1411,37.7164,0.0000
C00764=-48.058,10.965,6.549,179.5704,37.6118,0.0000
C00765=-48.078,11.826,6.572,-179.9860,37.4927,0.0000
C00766=-48.000,12.898,6.582,-179.4174,37.3356,0.0000
C00767=-47.771,14.270,6.588,-178.6689,37.1192,0.0000
C00768=-47.406,15.768,6.592,-177.8374,36.8604,0.0000
C00769=-46.944,17.193,6.597,-177.0366,36.5941,0.0000
C00770=-46.450,18.501,6.600,-176.3040,36.3310,0.0000
C00771=-45.928,19.763,6.600,150.4565,22.4702,0.0000
C00772=-45.352,21.037,6.597,150.6491,23.0906,0.0000
C00773=-44.670,22.372,6.592,150.8722,23.7547,0.0000
C00774=-43.870,23.689,6.588,151.1132,24.4328,0.0000
C00775=-43.061,24.821,6.582,151.3398,25.0326,0.0000
C00776=-42.359,25.634,6.572,151.5154,25.4837,0.0000
C00777=-41.735,26.229,6.549,151.6538,25.8335,0.0000
C00778=-41.112,26.810,6.517,151.7957,26.1655,0.0000
C00779=-40.393,27.570,6.484,151.9829,26.5514,0.0000
C00780=-39.419,28.746,6.458,152.2672,27.0624,0.0000
C00781=-38.009,30.513,6.447,152.6849,27.6993,0.0000
C00782=-36.374,32.441,6.446,152.5552,27.6539,0.0000
C00783=-34.464,34.464,6.447,150.9405,25.9058,0.0000
C00784=-32.441,36.374,6.446,149.4410,24.0949,0.0000
C00785=-30.513,38.009,6.447,149.4222,23.9726,0.0000
C00786=-28.746,39.419,6.458,150.0067,24.4819,0.0000
C00787=-27.570,40.393,6.484,150.4889,24.8471,0.0000
C00788=-26.810,41.112,6.517,150.8603,25.0994,0.0000
C00789=-26.229,41.735,6.549,151.1851,25.2997,0.0000
C00790=-25.634,42.359,6.572,151.5305,25.5009,0.0000
C00791=-24.821,43.061,6.582,151.9780,25.7576,0.0000
C00792=-23.689,43.870,6.588,152.5767,26.0924,0.0000
C00793=-22.372,44.670,6.592,153.2600,26.4565,0.0000
C00794=-21.037,45.352,6.597,153.9354,26.8006,0.0000
C00795=-19.763,45.928,6.600,154.5727,27.1065,0.0000
C00796=-18.501,46.450,6.600,143.6120,-2.9768,0.0000
C00797=-17.193,46.944,6.597,143.3692,-2.3789,0.0000
C00798=-15.768,47.406,6.592,143.1200,-1.7301,0.0000
C00799=-14.270,47.771,6.588,142.8734,-1.0614,0.0000
C00800=-12.898,48.000,6.582,142.6630,-0.4632,0.0000
C00801=-11.826,48.078,6.572,142.5073,-0.0111,0.0000
C00802=-10.965,48.058,6.549,142.3874,0.3403,0.0000
C00803=-10.113,48.028,6.517,142.2805,0.6794,0.0000
C00804=-9.067,48.057,6.484,142.1709,1.0857,0.0000
C00805=-7.547,48.199,6.458,142.0494,1.6430,0.0000
C00806=-5.301,48.453,6.447,141.9385,2.3719,0.0000
C00807=-2.781,48.660,6.446,141.8775,2.2645,0.0000
C00808=0.000,48.740,6.447,141.8391,0.0007,0.0000
C00809=0.000,47.885,8.473,141.4860,0.0006,0.0000
C00810=2.703,47.807,8.473,141.5254,-2.2766,0.0000
C00811=5.169,47.608,8.474,141.5829,-2.3278,0.0000
C00812=7.387,47.387,8.496,141.6890,-1.5573,0.0000
C00813=8.874,47.327,8.550,141.8073,-0.9859,0.0000
C00814=9.895,47.421,8.620,141.9163,-0.5760,0.0000
C00815=10.731,47.601,8.688,142.0259,-0.2352,0.0000
C00816=11.577,47.783,8.737,142.1505,0.1167,0.0000
C00817=12.629,47.854,8.761,142.3114,0.5694,0.0000
C00818=14.018,47.741,8.773,142.5329,1.1904,0.0000
C00819=15.568,47.442,8.783,142.7979,1.9032,0.0000
C00820=17.067,46.986,8.793,143.0698,2.6067,0.0000
C00821=18.458,46.467,8.799,143.3393,3.2621,0.0000
C00822=19.805,45.909,8.799,154.5425,-27.5000,0.0000
C00823=21.155,45.292,8.793,153.8387,-27.1665,0.0000
C00824=22.539,44.555,8.783,153.1029,-26.7940,0.0000
C00825=23.846,43.670,8.773,152.3713,-26.4064,0.0000
C00826=24.908,42.767,8.761,151.7460,-26.0598,0.0000
C00827=25.601,41.974,8.737,151.2929,-25.8052,0.0000
C00828=26.071,41.247,8.688,150.9426,-25.6060,0.0000
C00829=26.535,40.528,8.620,150.6140,-25.4055,0.0000
C00830=27.190,39.740,8.550,150.2402,-25.1493,0.0000
C00831=28.285,38.731,8.496,149.7510,-24.7701,0.0000
C00832=30.009,37.319,8.474,149.1426,-24.2237,0.0000
C00833=31.894,35.716,8.473,149.1268,-24.2992,0.0000
C00834=33.859,33.859,8.473,150.6322,-26.1248,0.0000
C00835=35.716,31.894,8.473,152.2537,-27.8837,0.0000
C00836=37.319,30.009,8.474,152.3406,-27.8875,0.0000
C00837=38.731,28.285,8.496,151.8903,-27.2197,0.0000
C00838=39.740,27.190,8.550,151.5947,-26.6991,0.0000
C00839=40.528,26.535,8.620,151.4056,-26.3103,0.0000
C00840=41.247,26.071,8.688,151.2658,-25.9751,0.0000
C00841=41.974,25.601,8.737,151.1323,-25.6218,0.0000
C00842=42.767,24.908,8.761,150.9622,-25.1666,0.0000
C00843=43.670,23.846,8.773,150.7315,-24.5415,0.0000
C00844=44.555,22.539,8.783,150.4787,-23.8170,0.0000
C00845=45.292,21.155,8.793,150.2407,-23.0953,0.0000
C00846=45.909,19.805,8.799,150.0346,-22.4126,0.0000
C00847=46.467,18.458,8.799,-175.9359,-36.5916,0.0000
C00848=46.986,17.067,8.793,-176.7404,-36.8857,0.0000
C00849=47.442,15.568,8.783,-177.6111,-37.1782,0.0000
C00850=47.741,14.018,8.773,-178.5003,-37.4576,0.0000
C00851=47.854,12.629,8.761,-179.2805,-37.6864,0.0000
C00852=47.783,11.577,8.737,-179.8523,-37.8494,0.0000
C00853=47.601,10.731,8.688,179.7016,-37.9737,0.0000
C00854=47.421,9.895,8.620,179.2683,-38.0814,0.0000
C00855=47.327,8.874,8.550,178.7457,-38.1860,0.0000
C00856=47.387,7.387,8.496,178.0156,-38.2943,0.0000
C00857=47.608,5.169,8.474,177.0300,-38.3797,0.0000
C00858=47.807,2.703,8.473,177.0930,-38.4386,0.0000
C00859=47.885,0.000,8.473,-179.9992,-38.5140,0.0000
C00860=47.807,-2.703,8.473,-177.0932,-38.4387,0.0000
C00861=47.608,-5.169,8.474,-177.0304,-38.3796,0.0000
C00862=47.387,-7.387,8.496,-178.0163,-38.2942,0.0000
C00863=47.327,-8.874,8.550,-178.7463,-38.1860,0.0000
C00864=47.421,-9.895,8.620,-179.2688,-38.0813,0.0000
C00865=47.601,-10.731,8.688,-179.7021,-37.9737,0.0000
C00866=47.783,-11.577,8.737,179.8519,-37.8494,0.0000
C00867=47.854,-12.629,8.761,179.2802,-37.6864,0.0000
C00868=47.741,-14.018,8.773,178.5002,-37.4576,0.0000
C00869=47.442,-15.568,8.783,177.6111,-37.1781,0.0000
C00870=46.986,-17.067,8.793,176.7404,-36.8856,0.0000
C00871=46.467,-18.458,8.799,175.9360,-36.5915,0.0000
C00872=45.909,-19.805,8.799,-150.0345,-22.4126,0.0000
C00873=45.292,-21.155,8.793,-150.2405,-23.0953,0.0000
C00874=44.555,-22.539,8.783,-150.4787,-23.8171,0.0000
C00875=43.670,-23.846,8.773,-150.7316,-24.5416,0.0000
C00876=42.767,-24.908,8.761,-150.9623,-25.1669,0.0000
C00877=41.974,-25.601,8.737,-151.1324,-25.6221,0.0000
C00878=41.247,-26.071,8.688,-151.2660,-25.9754,0.0000
C00879=40.528,-26.535,8.620,-151.4058,-26.3106,0.0000
C00880=39.740,-27.190,8.550,-151.5950,-26.6995,0.0000
C00881=38.731,-28.285,8.496,-151.8907,-27.2202,0.0000
C00882=37.319,-30.009,8.474,-152.3408,-27.8878,0.0000
C00883=35.716,-31.894,8.473,-152.2539,-27.8838,0.0000
C00884=33.859,-33.859,8.473,-150.6314,-26.1238,0.0000
C00885=31.894,-35.716,8.473,-149.1268,-24.2994,0.0000
C00886=30.009,-37.319,8.474,-149.1429,-24.2239,0.0000
C00887=28.285,-38.731,8.496,-149.7514,-24.7705,0.0000
C00888=27.190,-39.740,8.550,-150.2406,-25.1497,0.0000
C00889=26.535,-40.528,8.620,-150.6144,-25.4058,0.0000
C00890=26.071,-41.247,8.688,-150.9429,-25.6063,0.0000
C00891=25.601,-41.974,8.737,-151.2932,-25.8054,0.0000
C00892=24.908,-42.767,8.761,-151.7462,-26.0599,0.0000
C00893=23.846,-43.670,8.773,-152.3715,-26.4064,0.0000
C00894=22.539,-44.555,8.783,-153.1029,-26.7940,0.0000
C00895=21.155,-45.292,8.793,-153.8387,-27.1664,0.0000
C00896=19.805,-45.909,8.799,-154.5425,-27.4999,0.0000
C00897=18.458,-46.467,8.799,-143.3393,3.2621,0.0000
C00898=17.067,-46.986,8.793,-143.0698,2.6067,0.0000
C00899=15.568,-47.442,8.783,-142.7979,1.9032,0.0000
C00900=14.018,-47.741,8.773,-142.5329,1.1904,0.0000
C00901=12.629,-47.854,8.761,-142.3114,0.5694,0.0000
C00902=11.577,-47.783,8.737,-142.1505,0.1167,0.0000
C00903=10.731,-47.601,8.688,-142.0259,-0.2352,0.0000
C00904=9.895,-47.421,8.620,-141.9163,-0.5760,0.0000
C00905=8.874,-47.327,8.550,-141.8073,-0.9859,0.0000
C00906=7.387,-47.387,8.496,-141.6890,-1.5573,0.0000
C00907=5.169,-47.608,8.474,-141.5829,-2.3278,0.0000
C00908=2.703,-47.807,8.473,-141.5254,-2.2766,0.0000
C00909=0.000,-47.885,8.473,-141.4860,0.0006,0.0000
C00910=0.000,-47.885,8.473,-141.4860,0.0006,0.0000
C00911=-2.703,-47.807,8.473,-141.5254,2.2764,0.0000
C00912=-5.169,-47.608,8.474,-141.5829,2.3275,0.0000
C00913=-7.387,-47.387,8.496,-141.6891,1.5567,0.0000
C00914=-8.874,-47.327,8.550,-141.8073,0.9854,0.0000
C00915=-9.895,-47.421,8.620,-141.9164,0.5755,0.0000
C00916=-10.731,-47.601,8.688,-142.0259,0.2348,0.0000
C00917=-11.577,-47.783,8.737,-142.1505,-0.1170,0.0000
C00918=-12.629,-47.854,8.761,-142.3114,-0.5696,0.0000
C00919=-14.018,-47.741,8.773,-142.5330,-1.1905,0.0000
C00920=-15.568,-47.442,8.783,-142.7979,-1.9032,0.0000
C00921=-17.067,-46.986,8.793,-143.0699,-2.6066,0.0000
C00922=-18.458,-46.467,8.799,-143.3394,-3.2620,0.0000
C00923=-19.805,-45.909,8.799,-154.5425,27.5000,0.0000
C00924=-21.155,-45.292,8.793,-153.8387,27.1665,0.0000
C00925=-22.539,-44.555,8.783,-153.1029,26.7940,0.0000
C00926=-23.846,-43.670,8.773,-152.3713,26.4064,0.0000
C00927=-24.908,-42.767,8.761,-151.7460,26.0598,0.0000
C00928=-25.601,-41.974,8.737,-151.2929,25.8052,0.0000
C00929=-26.071,-41.247,8.688,-150.9426,25.6060,0.0000
C00930=-26.535,-40.528,8.620,-150.6140,25.4055,0.0000
C00931=-27.190,-39.740,8.550,-150.2402,25.1493,0.0000
C00932=-28.285,-38.731,8.496,-149.7510,24.7701,0.0000
C00933=-30.009,-37.319,8.474,-149.1426,24.2237,0.0000
C00934=-31.894,-35.716,8.473,-149.1268,24.2992,0.0000
C00935=-33.859,-33.859,8.473,-150.6322,26.1248,0.0000
C00936=-35.716,-31.894,8.473,-152.2537,27.8837,0.0000
C00937=-37.319,-30.009,8.474,-152.3406,27.8875,0.0000
C00938=-38.731,-28.285,8.496,-151.8903,27.2197,0.0000
C00939=-39.740,-27.190,8.550,-151.5947,26.6991,0.0000
C00940=-40.528,-26.535,8.620,-151.4056,26.3103,0.0000
C00941=-41.247,-26.071,8.688,-151.2658,25.9751,0.0000
C00942=-41.974,-25.601,8.737,-151.1323,25.6218,0.0000
C00943=-42.767,-24.908,8.761,-150.9622,25.1666,0.0000
C00944=-43.670,-23.846,8.773,-150.7315,24.5415,0.0000
C00945=-44.555,-22.539,8.783,-150.4787,23.8170,0.0000
C00946=-45.292,-21.155,8.793,-150.2407,23.0953,0.0000
C00947=-45.909,-19.805,8.799,-150.0346,22.4126,0.0000
C00948=-46.467,-18.458,8.799,175.9359,36.5916,0.0000
C00949=-46.986,-17.067,8.793,176.7404,36.8857,0.0000
C00950=-47.442,-15.568,8.783,177.6111,37.1782,0.0000
C00951=-47.741,-14.018,8.773,178.5003,37.4576,0.0000
C00952=-47.854,-12.629,8.761,179.2805,37.6864,0.0000
C00953=-47.783,-11.577,8.737,179.8523,37.8494,0.0000
C00954=-47.601,-10.731,8.688,-179.7016,37.9737,0.0000
C00955=-47.421,-9.895,8.620,-179.2683,38.0814,0.0000
C00956=-47.327,-8.874,8.550,-178.7457,38.1860,0.0000
C00957=-47.387,-7.387,8.496,-178.0156,38.2943,0.0000
C00958=-47.608,-5.169,8.474,-177.0300,38.3797,0.0000
C00959=-47.807,-2.703,8.473,-177.0930,38.4386,0.0000
C00960=-47.885,0.000,8.473,179.9992,38.5140,0.0000
C00961=-47.807,2.703,8.473,177.0932,38.4387,0.0000
C00962=-47.608,5.169,8.474,177.0304,38.3796,0.0000
C00963=-47.387,7.387,8.496,178.0163,38.2942,0.0000
C00964=-47.327,8.874,8.550,178.7463,38.1860,0.0000
C00965=-47.421,9.895,8.620,179.2688,38.0813,0.0000
C00966=-47.601,10.731,8.688,179.7021,37.9737,0.0000
C00967=-47.783,11.577,8.737,-179.8519,37.8494,0.0000
C00968=-47.854,12.629,8.761,-179.2802,37.6864,0.0000
C00969=-47.741,14.018,8.773,-178.5002,37.4576,0.0000
C00970=-47.442,15.568,8.783,-177.6111,37.1781,0.0000
C00971=-46.986,17.067,8.793,-176.7404,36.8856,0.0000
C00972=-46.467,18.458,8.799,-175.9360,36.5915,0.0000
C00973=-45.909,19.805,8.799,150.0345,22.4126,0.0000
C00974=-45.292,21.155,8.793,150.2405,23.0953,0.0000
C00975=-44.555,22.539,8.783,150.4787,23.8171,0.0000
C00976=-43.670,23.846,8.773,150.7316,24.5416,0.0000
C00977=-42.767,24.908,8.761,150.9623,25.1669,0.0000
C00978=-41.974,25.601,8.737,151.1324,25.6221,0.0000
C00979=-41.247,26.071,8.688,151.2660,25.9754,0.0000
C00980=-40.528,26.535,8.620,151.4058,26.3106,0.0000
C00981=-39.740,27.190,8.550,151.5950,26.6995,0.0000
C00982=-38.731,28.285,8.496,151.8907,27.2202,0.0000
C00983=-37.319,30.009,8.474,152.3408,27.8878,0.0000
C00984=-35.716,31.894,8.473,152.2539,27.8838,0.0000
C00985=-33.859,33.859,8.473,150.6314,26.1238,0.0000
C00986=-31.894,35.716,8.473,149.1268,24.2994,0.0000
C00987=-30.009,37.319,8.474,149.1429,24.2239,0.0000
C00988=-28.285,38.731,8.496,149.7514,24.7705,0.0000
C00989=-27.190,39.740,8.550,150.2406,25.1497,0.0000
C00990=-26.535,40.528,8.620,150.6144,25.4058,0.0000
C00991=-26.071,41.247,8.688,150.9429,25.6063,0.0000
C00992=-25.601,41.974,8.737,151.2932,25.8054,0.0000
C00993=-24.908,42.767,8.761,151.7462,26.0599,0.0000
C00994=-23.846,43.670,8.773,152.3715,26.4064,0.0000
C00995=-22.539,44.555,8.783,153.1029,26.7940,0.0000
C00996=-21.155,45.292,8.793,153.8387,27.1664,0.0000
C00997=-19.805,45.909,8.799,154.5425,27.4999,0.0000
C00998=-18.458,46.467,8.799,143.3394,-3.2620,0.0000
C00999=-17.067,46.986,8.793,143.0699,-2.6066,0.0000
C01000=-15.568,47.442,8.783,142.7979,-1.9032,0.0000
C01001=-14.018,47.741,8.773,142.5330,-1.1905,0.0000
C01002=-12.629,47.854,8.761,142.3114,-0.5696,0.0000
C01003=-11.577,47.783,8.737,142.1505,-0.1170,0.0000
C01004=-10.731,47.601,8.688,142.0259,0.2348,0.0000
C01005=-9.895,47.421,8.620,141.9164,0.5755,0.0000
C01006=-8.874,47.327,8.550,141.8073,0.9854,0.0000
C01007=-7.387,47.387,8.496,141.6891,1.5567,0.0000
C01008=-5.169,47.608,8.474,141.5829,2.3275,0.0000
C01009=-2.703,47.807,8.473,141.5254,2.2764,0.0000
C01010=0.000,47.885,8.473,141.4860,0.0006,0.0000
C01011=0.000,46.884,10.433,141.2072,0.0005,0.0000
C01012=2.611,46.810,10.432,141.2474,-2.2809,0.0000
C01013=5.015,46.620,10.433,141.3016,-2.2862,0.0000
C01014=7.199,46.436,10.471,141.4028,-1.4819,0.0000
C01015=8.646,46.466,10.562,141.5160,-0.9031,0.0000
C01016=9.635,46.699,10.682,141.6215,-0.4951,0.0000
C01017=10.451,47.054,10.800,141.7298,-0.1569,0.0000
C01018=11.278,47.426,10.887,141.8551,0.1911,0.0000
C01019=12.303,47.677,10.929,142.0174,0.6393,0.0000
C01020=13.711,47.704,10.951,142.2479,1.2830,0.0000
C01021=15.325,47.486,10.969,142.5316,2.0451,0.0000
C01022=16.914,47.036,10.987,142.8296,2.8123,0.0000
C01023=18.406,46.487,10.998,143.1313,3.5354,0.0000
C01024=19.856,45.886,10.998,154.5596,-27.8430,0.0000
C01025=21.300,45.220,10.987,153.7772,-27.4777,0.0000
C01026=22.741,44.414,10.969,152.9716,-27.0720,0.0000
C01027=24.036,43.427,10.951,152.1878,-26.6569,0.0000
C01028=25.013,42.412,10.929,151.5381,-26.2974,0.0000
C01029=25.561,41.510,10.887,151.0864,-26.0466,0.0000
C01030=25.882,40.662,10.800,150.7377,-25.8505,0.0000
C01031=26.208,39.834,10.682,150.4117,-25.6507,0.0000
C01032=26.743,38.970,10.562,150.0419,-25.3933,0.0000
C01033=27.744,37.925,10.471,149.5519,-25.0044,0.0000
C01034=29.419,36.512,10.433,148.9252,-24.4274,0.0000
C01035=31.253,34.946,10.432,148.8814,-24.4644,0.0000
C01036=33.152,33.152,10.433,150.3872,-26.2962,0.0000
C01037=34.946,31.253,10.432,152.0113,-28.0609,0.0000
C01038=36.512,29.419,10.433,152.0629,-28.0310,0.0000
C01039=37.925,27.744,10.471,151.5857,-27.3390,0.0000
C01040=38.970,26.743,10.562,151.2816,-26.8151,0.0000
C01041=39.834,26.208,10.682,151.0914,-26.4296,0.0000
C01042=40.662,25.882,10.800,150.9530,-26.0969,0.0000
C01043=41.510,25.561,10.887,150.8235,-25.7459,0.0000
C01044=42.412,25.013,10.929,150.6589,-25.2931,0.0000
C01045=43.427,24.036,10.951,150.4220,-24.6440,0.0000
C01046=44.414,22.741,10.969,150.1538,-23.8686,0.0000
C01047=45.220,21.300,10.987,149.8976,-23.0800,0.0000
C01048=45.886,19.856,10.998,149.6760,-22.3238,0.0000
C01049=46.487,18.406,10.998,-175.5839,-36.7870,0.0000
C01050=47.036,16.914,10.987,-176.4723,-37.1181,0.0000
C01051=47.486,15.325,10.969,-177.4239,-37.4404,0.0000
C01052=47.704,13.711,10.951,-178.3775,-37.7409,0.0000
C01053=47.677,12.303,10.929,-179.1890,-37.9798,0.0000
C01054=47.426,11.278,10.887,-179.7570,-38.1447,0.0000
C01055=47.054,10.451,10.800,179.8002,-38.2700,0.0000
C01056=46.699,9.635,10.682,179.3685,-38.3768,0.0000
C01057=46.466,8.646,10.562,178.8464,-38.4783,0.0000
C01058=46.436,7.199,10.471,178.1042,-38.5819,0.0000
C01059=46.620,5.015,10.433,177.0717,-38.6619,0.0000
C01060=46.810,2.611,10.432,177.0762,-38.7162,0.0000
C01061=46.884,0.000,10.433,-179.9994,-38.7928,0.0000
C01062=46.810,-2.611,10.432,-177.0764,-38.7163,0.0000
C01063=46.620,-5.015,10.433,-177.0721,-38.6619,0.0000
C01064=46.436,-7.199,10.471,-178.1049,-38.5818,0.0000
C01065=46.466,-8.646,10.562,-178.8470,-38.4783,0.0000
C01066=46.699,-9.635,10.682,-179.3691,-38.3768,0.0000
C01067=47.054,-10.451,10.800,-179.8007,-38.2700,0.0000
C01068=47.426,-11.278,10.887,179.7566,-38.1446,0.0000
C01069=47.677,-12.303,10.929,179.1887,-37.9797,0.0000
C01070=47.704,-13.711,10.951,178.3773,-37.7409,0.0000
C01071=47.486,-15.325,10.969,177.4239,-37.4404,0.0000
C01072=47.036,-16.914,10.987,176.4724,-37.1180,0.0000
C01073=46.487,-18.406,10.998,175.5840,-36.7869,0.0000
C01074=45.886,-19.856,10.998,-149.6759,-22.3238,0.0000
C01075=45.220,-21.300,10.987,-149.8975,-23.0800,0.0000
C01076=44.414,-22.741,10.969,-150.1538,-23.8687,0.0000
C01077=43.427,-24.036,10.951,-150.4220,-24.6442,0.0000
C01078=42.412,-25.013,10.929,-150.6590,-25.2933,0.0000
C01079=41.510,-25.561,10.887,-150.8237,-25.7462,0.0000
C01080=40.662,-25.882,10.800,-150.9532,-26.0972,0.0000
C01081=39.834,-26.208,10.682,-151.0916,-26.4299,0.0000
C01082=38.970,-26.743,10.562,-151.2819,-26.8156,0.0000
C01083=37.925,-27.744,10.471,-151.5860,-27.3394,0.0000
C01084=36.512,-29.419,10.433,-152.0631,-28.0313,0.0000
C01085=34.946,-31.253,10.432,-152.0115,-28.0610,0.0000
C01086=33.152,-33.152,10.433,-150.3866,-26.2955,0.0000
C01087=31.253,-34.946,10.432,-148.8815,-24.4646,0.0000
C01088=29.419,-36.512,10.433,-148.9255,-24.4276,0.0000
C01089=27.744,-37.925,10.471,-149.5524,-25.0048,0.0000
C01090=26.743,-38.970,10.562,-150.0423,-25.3937,0.0000
C01091=26.208,-39.834,10.682,-150.4121,-25.6510,0.0000
C01092=25.882,-40.662,10.800,-150.7380,-25.8507,0.0000
C01093=25.561,-41.510,10.887,-151.0867,-26.0469,0.0000
C01094=25.013,-42.412,10.929,-151.5383,-26.2976,0.0000
C01095=24.036,-43.427,10.951,-152.1880,-26.6570,0.0000
C01096=22.741,-44.414,10.969,-152.9717,-27.0720,0.0000
C01097=21.300,-45.220,10.987,-153.7772,-27.4776,0.0000
C01098=19.856,-45.886,10.998,-154.5596,-27.8428,0.0000
C01099=18.406,-46.487,10.998,-143.1313,3.5354,0.0000
C01100=16.914,-47.036,10.987,-142.8296,2.8123,0.0000
C01101=15.325,-47.486,10.969,-142.5316,2.0451,0.0000
C01102=13.711,-47.704,10.951,-142.2479,1.2830,0.0000
C01103=12.303,-47.677,10.929,-142.0174,0.6393,0.0000
C01104=11.278,-47.426,10.887,-141.8551,0.1911,0.0000
C01105=10.451,-47.054,10.800,-141.7298,-0.1569,0.0000
C01106=9.635,-46.699,10.682,-141.6215,-0.4951,0.0000
C01107=8.646,-46.466,10.562,-141.5160,-0.9031,0.0000
C01108=7.199,-46.436,10.471,-141.4028,-1.4819,0.0000
C01109=5.015,-46.620,10.433,-141.3016,-2.2862,0.0000
C01110=2.611,-46.810,10.432,-141.2474,-2.2809,0.0000
C01111=0.000,-46.884,10.433,-141.2072,0.0005,0.0000
C01112=0.000,-46.884,10.433,-141.2072,0.0005,0.0000
C01113=-2.611,-46.810,10.432,-141.2473,2.2807,0.0000
C01114=-5.015,-46.620,10.433,-141.3016,2.2858,0.0000
C01115=-7.199,-46.436,10.471,-141.4029,1.4814,0.0000
C01116=-8.646,-46.466,10.562,-141.5161,0.9026,0.0000
C01117=-9.635,-46.699,10.682,-141.6215,0.4946,0.0000
C01118=-10.451,-47.054,10.800,-141.7298,0.1565,0.0000
C01119=-11.278,-47.426,10.887,-141.8551,-0.1914,0.0000
C01120=-12.303,-47.677,10.929,-142.0175,-0.6395,0.0000
C01121=-13.711,-47.704,10.951,-142.2480,-1.2831,0.0000
C01122=-15.325,-47.486,10.969,-142.5317,-2.0452,0.0000
C01123=-16.914,-47.036,10.987,-142.8297,-2.8122,0.0000
C01124=-18.406,-46.487,10.998,-143.1313,-3.5354,0.0000
C01125=-19.856,-45.886,10.998,-154.5596,27.8430,0.0000
C01126=-21.300,-45.220,10.987,-153.7772,27.4777,0.0000
C01127=-22.741,-44.414,10.969,-152.9716,27.0720,0.0000
C01128=-24.036,-43.427,10.951,-152.1878,26.6569,0.0000
C01129=-25.013,-42.412,10.929,-151.5381,26.2974,0.0000
C01130=-25.561,-41.510,10.887,-151.0864,26.0466,0.0000
C01131=-25.882,-40.662,10.800,-150.7377,25.8505,0.0000
C01132=-26.208,-39.834,10.682,-150.4117,25.6507,0.0000
C01133=-26.743,-38.970,10.562,-150.0419,25.3933,0.0000
C01134=-27.744,-37.925,10.471,-149.5519,25.0044,0.0000
C01135=-29.419,-36.512,10.433,-148.9252,24.4274,0.0000
C01136=-31.253,-34.946,10.432,-148.8814,24.4644,0.0000
C01137=-33.152,-33.152,10.433,-150.3872,26.2962,0.0000
C01138=-34.946,-31.253,10.432,-152.0113,28.0609,0.0000
C01139=-36.512,-29.419,10.433,-152.0629,28.0310,0.0000
C01140=-37.925,-27.744,10.471,-151.5857,27.3390,0.0000
C01141=-38.970,-26.743,10.562,-151.2816,26.8151,0.0000
C01142=-39.834,-26.208,10.682,-151.0914,26.4296,0.0000
C01143=-40.662,-25.882,10.800,-150.9530,26.0969,0.0000
C01144=-41.510,-25.561,10.887,-150.8235,25.7459,0.0000
C01145=-42.412,-25.013,10.929,-150.6589,25.2931,0.0000
C01146=-43.427,-24.036,10.951,-150.4220,24.6440,0.0000
C01147=-44.414,-22.741,10.969,-150.1538,23.8686,0.0000
C01148=-45.220,-21.300,10.987,-149.8976,23.0800,0.0000
C01149=-45.886,-19.856,10.998,-149.6760,22.3238,0.0000
C01150=-46.487,-18.406,10.998,175.5839,36.7870,0.0000
C01151=-47.036,-16.914,10.987,176.4723,37.1181,0.0000
C01152=-47.486,-15.325,10.969,177.4239,37.4404,0.0000
C01153=-47.704,-13.711,10.951,178.3775,37.7409,0.0000
C01154=-47.677,-12.303,10.929,179.1890,37.9798,0.0000
C01155=-47.426,-11.278,10.887,179.7570,38.1447,0.0000
C01156=-47.054,-10.451,10.800,-179.8002,38.2700,0.0000
C01157=-46.699,-9.635,10.682,-179.3685,38.3768,0.0000
C01158=-46.466,-8.646,10.562,-178.8464,38.4783,0.0000
C01159=-46.436,-7.199,10.471,-178.1042,38.5819,0.0000
C01160=-46.620,-5.015,10.433,-177.0717,38.6619,0.0000
C01161=-46.810,-2.611,10.432,-177.0762,38.7162,0.0000
C01162=-46.884,0.000,10.433,179.9994,38.7928,0.0000
C01163=-46.810,2.611,10.432,177.0764,38.7163,0.0000
C01164=-46.620,5.015,10.433,177.0721,38.6619,0.0000
C01165=-46.436,7.199,10.471,178.1049,38.5818,0.0000
C01166=-46.466,8.646,10.562,178.8470,38.4783,0.0000
C01167=-46.699,9.635,10.682,179.3691,38.3768,0.0000
C01168=-47.054,10.451,10.800,179.8007,38.2700,0.0000
C01169=-47.426,11.278,10.887,-179.7566,38.1446,0.0000
C01170=-47.677,12.303,10.929,-179.1887,37.9797,0.0000
C01171=-47.704,13.711,10.951,-178.3773,37.7409,0.0000
C01172=-47.486,15.325,10.969,-177.4239,37.4404,0.0000
C01173=-47.036,16.914,10.987,-176.4724,37.1180,0.0000
C01174=-46.487,18.406,10.998,-175.5840,36.7869,0.0000
C01175=-45.886,19.856,10.998,149.6759,22.3238,0.0000
C01176=-45.220,21.300,10.987,149.8975,23.0800,0.0000
C01177=-44.414,22.741,10.969,150.1538,23.8687,0.0000
C01178=-43.427,24.036,10.951,150.4220,24.6442,0.0000
C01179=-42.412,25.013,10.929,150.6590,25.2933,0.0000
C01180=-41.510,25.561,10.887,150.8237,25.7462,0.0000
C01181=-40.662,25.882,10.800,150.9532,26.0972,0.0000
C01182=-39.834,26.208,10.682,151.0916,26.4299,0.0000
C01183=-38.970,26.743,10.562,151.2819,26.8156,0.0000
C01184=-37.925,27.744,10.471,151.5860,27.3394,0.0000
C01185=-36.512,29.419,10.433,152.0631,28.0313,0.0000
C01186=-34.946,31.253,10.432,152.0115,28.0610,0.0000
C01187=-33.152,33.152,10.433,150.3866,26.2955,0.0000
C01188=-31.253,34.946,10.432,148.8815,24.4646,0.0000
C01189=-29.419,36.512,10.433,148.9255,24.4276,0.0000
C01190=-27.744,37.925,10.471,149.5524,25.0048,0.0000
C01191=-26.743,38.970,10.562,150.0423,25.3937,0.0000
C01192=-26.208,39.834,10.682,150.4121,25.6510,0.0000
C01193=-25.882,40.662,10.800,150.7380,25.8507,0.0000
C01194=-25.561,41.510,10.887,151.0867,26.0469,0.0000
C01195=-25.013,42.412,10.929,151.5383,26.2976,0.0000
C01196=-24.036,43.427,10.951,152.1880,26.6570,0.0000
C01197=-22.741,44.414,10.969,152.9717,27.0720,0.0000
C01198=-21.300,45.220,10.987,153.7772,27.4776,0.0000
C01199=-19.856,45.886,10.998,154.5596,27.8428,0.0000
C01200=-18.406,46.487,10.998,143.1313,-3.5354,0.0000
C01201=-16.914,47.036,10.987,142.8297,-2.8122,0.0000
C01202=-15.325,47.486,10.969,142.5317,-2.0452,0.0000
C01203=-13.711,47.704,10.951,142.2480,-1.2831,0.0000
C01204=-12.303,47.677,10.929,142.0175,-0.6395,0.0000
C01205=-11.278,47.426,10.887,141.8551,-0.1914,0.0000
C01206=-10.451,47.054,10.800,141.7298,0.1565,0.0000
C01207=-9.635,46.699,10.682,141.6215,0.4946,0.0000
C01208=-8.646,46.466,10.562,141.5161,0.9026,0.0000
C01209=-7.199,46.436,10.471,141.4029,1.4814,0.0000
C01210=-5.015,46.620,10.433,141.3016,2.2858,0.0000
C01211=-2.611,46.810,10.432,141.2473,2.2807,0.0000
C01212=0.000,46.884,10.433,141.2072,0.0005,0.0000
C01213=0.000,45.772,12.331,140.9966,0.0004,0.0000
C01214=2.510,45.702,12.329,141.0372,-2.2783,0.0000
C01215=4.844,45.521,12.332,141.0883,-2.2480,0.0000
C01216=6.990,45.375,12.387,141.1844,-1.4176,0.0000
C01217=8.390,45.503,12.523,141.2910,-0.8370,0.0000
C01218=9.343,45.885,12.705,141.3901,-0.4361,0.0000
C01219=10.132,46.432,12.887,141.4933,-0.1043,0.0000
C01220=10.935,47.018,13.022,141.6148,0.2360,0.0000
C01221=11.930,47.474,13.088,141.7741,0.6752,0.0000
C01222=13.360,47.661,13.123,142.0105,1.3418,0.0000
C01223=15.047,47.537,13.151,142.3124,2.1587,0.0000
C01224=16.738,47.094,13.179,142.6394,2.9983,0.0000
C01225=18.347,46.510,13.197,142.9784,3.7988,0.0000
C01226=19.915,45.860,13.197,154.6177,-28.1429,0.0000
C01227=21.465,45.136,13.179,153.7449,-27.7421,0.0000
C01228=22.974,44.253,13.151,152.8609,-27.2982,0.0000
C01229=24.255,43.149,13.123,152.0215,-26.8512,0.0000
C01230=25.133,42.005,13.088,151.3501,-26.4767,0.0000
C01231=25.514,40.979,13.022,150.9071,-26.2305,0.0000
C01232=25.668,39.997,12.887,150.5667,-26.0376,0.0000
C01233=25.839,39.052,12.705,150.2493,-25.8394,0.0000
C01234=26.243,38.108,12.523,149.8897,-25.5834,0.0000
C01235=27.143,37.028,12.387,149.4040,-25.1884,0.0000
C01236=28.763,35.614,12.332,148.7642,-24.5868,0.0000
C01237=30.541,34.091,12.329,148.6994,-24.5936,0.0000
C01238=32.366,32.366,12.331,150.2016,-26.4256,0.0000
C01239=34.091,30.541,12.329,151.8234,-28.1900,0.0000
C01240=35.614,28.763,12.332,151.8472,-28.1343,0.0000
C01241=37.028,27.143,12.387,151.3481,-27.4243,0.0000
C01242=38.108,26.243,12.523,151.0376,-26.9026,0.0000
C01243=39.052,25.839,12.705,150.8475,-26.5263,0.0000
C01244=39.997,25.668,12.887,150.7096,-26.2015,0.0000
C01245=40.979,25.514,13.022,150.5827,-25.8587,0.0000
C01246=42.005,25.133,13.088,150.4222,-25.4146,0.0000
C01247=43.149,24.255,13.123,150.1760,-24.7435,0.0000
C01248=44.253,22.974,13.151,149.8883,-23.9131,0.0000
C01249=45.136,21.465,13.179,149.6105,-23.0490,0.0000
C01250=45.860,19.915,13.197,149.3717,-22.2085,0.0000
C01251=46.510,18.347,13.197,-175.2460,-36.9267,0.0000
C01252=47.094,16.738,13.179,-176.2297,-37.3007,0.0000
C01253=47.537,15.047,13.151,-177.2729,-37.6562,0.0000
C01254=47.661,13.360,13.123,-178.2977,-37.9773,0.0000
C01255=47.474,11.930,13.088,-179.1406,-38.2227,0.0000
C01256=47.018,10.935,13.022,-179.6989,-38.3848,0.0000
C01257=46.432,10.132,12.887,179.8667,-38.5066,0.0000
C01258=45.885,9.343,12.705,179.4420,-38.6086,0.0000
C01259=45.503,8.390,12.523,178.9275,-38.7041,0.0000
C01260=45.375,6.990,12.387,178.1808,-38.8015,0.0000
C01261=45.521,4.844,12.332,177.1119,-38.8762,0.0000
C01262=45.702,2.510,12.329,177.0709,-38.9262,0.0000
C01263=45.772,0.000,12.331,-179.9995,-39.0034,0.0000
C01264=45.702,-2.510,12.329,-177.0712,-38.9263,0.0000
C01265=45.521,-4.844,12.332,-177.1124,-38.8761,0.0000
C01266=45.375,-6.990,12.387,-178.1815,-38.8014,0.0000
C01267=45.503,-8.390,12.523,-178.9281,-38.7041,0.0000
C01268=45.885,-9.343,12.705,-179.4425,-38.6085,0.0000
C01269=46.432,-10.132,12.887,-179.8672,-38.5065,0.0000
C01270=47.018,-10.935,13.022,179.6984,-38.3847,0.0000
C01271=47.474,-11.930,13.088,179.1402,-38.2227,0.0000
C01272=47.661,-13.360,13.123,178.2975,-37.9772,0.0000
C01273=47.537,-15.047,13.151,177.2728,-37.6561,0.0000
C01274=47.094,-16.738,13.179,176.2297,-37.3006,0.0000
C01275=46.510,-18.347,13.197,175.2461,-36.9267,0.0000
C01276=45.860,-19.915,13.197,-149.3716,-22.2085,0.0000
C01277=45.136,-21.465,13.179,-149.6105,-23.0490,0.0000
C01278=44.253,-22.974,13.151,-149.8884,-23.9131,0.0000
C01279=43.149,-24.255,13.123,-150.1761,-24.7437,0.0000
C01280=42.005,-25.133,13.088,-150.4224,-25.4148,0.0000
C01281=40.979,-25.514,13.022,-150.5829,-25.8590,0.0000
C01282=39.997,-25.668,12.887,-150.7099,-26.2019,0.0000
C01283=39.052,-25.839,12.705,-150.8477,-26.5266,0.0000
C01284=38.108,-26.243,12.523,-151.0379,-26.9030,0.0000
C01285=37.028,-27.143,12.387,-151.3484,-27.4248,0.0000
C01286=35.614,-28.763,12.332,-151.8475,-28.1346,0.0000
C01287=34.091,-30.541,12.329,-151.8236,-28.1901,0.0000
C01288=32.366,-32.366,12.331,-150.2011,-26.4249,0.0000
C01289=30.541,-34.091,12.329,-148.6994,-24.5938,0.0000
C01290=28.763,-35.614,12.332,-148.7645,-24.5871,0.0000
C01291=27.143,-37.028,12.387,-149.4044,-25.1888,0.0000
C01292=26.243,-38.108,12.523,-149.8901,-25.5837,0.0000
C01293=25.839,-39.052,12.705,-150.2497,-25.8397,0.0000
C01294=25.668,-39.997,12.887,-150.5670,-26.0379,0.0000
C01295=25.514,-40.979,13.022,-150.9073,-26.2307,0.0000
C01296=25.133,-42.005,13.088,-151.3503,-26.4769,0.0000
C01297=24.255,-43.149,13.123,-152.0216,-26.8513,0.0000
C01298=22.974,-44.253,13.151,-152.8610,-27.2983,0.0000
C01299=21.465,-45.136,13.179,-153.7450,-27.7420,0.0000
C01300=19.915,-45.860,13.197,-154.6177,-28.1428,0.0000
C01301=18.347,-46.510,13.197,-142.9784,3.7988,0.0000
C01302=16.738,-47.094,13.179,-142.6394,2.9983,0.0000
C01303=15.047,-47.537,13.151,-142.3124,2.1587,0.0000
C01304=13.360,-47.661,13.123,-142.0105,1.3418,0.0000
C01305=11.930,-47.474,13.088,-141.7741,0.6752,0.0000
C01306=10.935,-47.018,13.022,-141.6148,0.2360,0.0000
C01307=10.132,-46.432,12.887,-141.4933,-0.1043,0.0000
C01308=9.343,-45.885,12.705,-141.3901,-0.4361,0.0000
C01309=8.390,-45.503,12.523,-141.2910,-0.8370,0.0000
C01310=6.990,-45.375,12.387,-141.1844,-1.4176,0.0000
C01311=4.844,-45.521,12.332,-141.0883,-2.2480,0.0000
C01312=2.510,-45.702,12.329,-141.0372,-2.2783,0.0000
C01313=0.000,-45.772,12.331,-140.9966,0.0004,0.0000
C01314=0.000,-45.772,12.331,-140.9966,0.0004,0.0000
C01315=-2.510,-45.702,12.329,-141.0371,2.2781,0.0000
C01316=-4.844,-45.521,12.332,-141.0883,2.2477,0.0000
C01317=-6.990,-45.375,12.387,-141.1845,1.4171,0.0000
C01318=-8.390,-45.503,12.523,-141.2910,0.8365,0.0000
C01319=-9.343,-45.885,12.705,-141.3902,0.4356,0.0000
C01320=-10.132,-46.432,12.887,-141.4934,0.1039,0.0000
C01321=-10.935,-47.018,13.022,-141.6149,-0.2364,0.0000
C01322=-11.930,-47.474,13.088,-141.7742,-0.6754,0.0000
C01323=-13.360,-47.661,13.123,-142.0105,-1.3420,0.0000
C01324=-15.047,-47.537,13.151,-142.3125,-2.1588,0.0000
C01325=-16.738,-47.094,13.179,-142.6395,-2.9983,0.0000
C01326=-18.347,-46.510,13.197,-142.9785,-3.7987,0.0000
C01327=-19.915,-45.860,13.197,-154.6177,28.1429,0.0000
C01328=-21.465,-45.136,13.179,-153.7449,27.7421,0.0000
C01329=-22.974,-44.253,13.151,-152.8609,27.2982,0.0000
C01330=-24.255,-43.149,13.123,-152.0215,26.8512,0.0000
C01331=-25.133,-42.005,13.088,-151.3501,26.4767,0.0000
C01332=-25.514,-40.979,13.022,-150.9071,26.2305,0.0000
C01333=-25.668,-39.997,12.887,-150.5667,26.0376,0.0000
C01334=-25.839,-39.052,12.705,-150.2493,25.8394,0.0000
C01335=-26.243,-38.108,12.523,-149.8897,25.5834,0.0000
C01336=-27.143,-37.028,12.387,-149.4040,25.1884,0.0000
C01337=-28.763,-35.614,12.332,-148.7642,24.5868,0.0000
C01338=-30.541,-34.091,12.329,-148.6994,24.5936,0.0000
C01339=-32.366,-32.366,12.331,-150.2016,26.4256,0.0000
C01340=-34.091,-30.541,12.329,-151.8234,28.1900,0.0000
C01341=-35.614,-28.763,12.332,-151.8472,28.1343,0.0000
C01342=-37.028,-27.143,12.387,-151.3481,27.4243,0.0000
C01343=-38.108,-26.243,12.523,-151.0376,26.9026,0.0000
C01344=-39.052,-25.839,12.705,-150.8475,26.5263,0.0000
C01345=-39.997,-25.668,12.887,-150.7096,26.2015,0.0000
C01346=-40.979,-25.514,13.022,-150.5827,25.8587,0.0000
C01347=-42.005,-25.133,13.088,-150.4222,25.4146,0.0000
C01348=-43.149,-24.255,13.123,-150.1760,24.7435,0.0000
C01349=-44.253,-22.974,13.151,-149.8883,23.9131,0.0000
C01350=-45.136,-21.465,13.179,-149.6105,23.0490,0.0000
C01351=-45.860,-19.915,13.197,-149.3717,22.2085,0.0000
C01352=-46.510,-18.347,13.197,175.2460,36.9267,0.0000
C01353=-47.094,-16.738,13.179,176.2297,37.3007,0.0000
C01354=-47.537,-15.047,13.151,177.2729,37.6562,0.0000
C01355=-47.661,-13.360,13.123,178.2977,37.9773,0.0000
C01356=-47.474,-11.930,13.088,179.1406,38.2227,0.0000
C01357=-47.018,-10.935,13.022,179.6989,38.3848,0.0000
C01358=-46.432,-10.132,12.887,-179.8667,38.5066,0.0000
C01359=-45.885,-9.343,12.705,-179.4420,38.6086,0.0000
C01360=-45.503,-8.390,12.523,-178.9275,38.7041,0.0000
C01361=-45.375,-6.990,12.387,-178.1808,38.8015,0.0000
C01362=-45.521,-4.844,12.332,-177.1119,38.8762,0.0000
C01363=-45.702,-2.510,12.329,-177.0709,38.9262,0.0000
C01364=-45.772,0.000,12.331,179.9995,39.0034,0.0000
C01365=-45.702,2.510,12.329,177.0712,38.9263,0.0000
C01366=-45.521,4.844,12.332,177.1124,38.8761,0.0000
C01367=-45.375,6.990,12.387,178.1815,38.8014,0.0000
C01368=-45.503,8.390,12.523,178.9281,38.7041,0.0000
C01369=-45.885,9.343,12.705,179.4425,38.6085,0.0000
C01370=-46.432,10.132,12.887,179.8672,38.5065,0.0000
C01371=-47.018,10.935,13.022,-179.6984,38.3847,0.0000
C01372=-47.474,11.930,13.088,-179.1402,38.2227,0.0000
C01373=-47.661,13.360,13.123,-178.2975,37.9772,0.0000
C01374=-47.537,15.047,13.151,-177.2728,37.6561,0.0000
C01375=-47.094,16.738,13.179,-176.2297,37.3006,0.0000
C01376=-46.510,18.347,13.197,-175.2461,36.9267,0.0000
C01377=-45.860,19.915,13.197,149.3716,22.2085,0.0000
C01378=-45.136,21.465,13.179,149.6105,23.0490,0.0000
C01379=-44.253,22.974,13.151,149.8884,23.9131,0.0000
C01380=-43.149,24.255,13.123,150.1761,24.7437,0.0000
C01381=-42.005,25.133,13.088,150.4224,25.4148,0.0000
C01382=-40.979,25.514,13.022,150.5829,25.8590,0.0000
C01383=-39.997,25.668,12.887,150.7099,26.2019,0.0000
C01384=-39.052,25.839,12.705,150.8477,26.5266,0.0000
C01385=-38.108,26.243,12.523,151.0379,26.9030,0.0000
C01386=-37.028,27.143,12.387,151.3484,27.4248,0.0000
C01387=-35.614,28.763,12.332,151.8475,28.1346,0.0000
C01388=-34.091,30.541,12.329,151.8236,28.1901,0.0000
C01389=-32.366,32.366,12.331,150.2011,26.4249,0.0000
C01390=-30.541,34.091,12.329,148.6994,24.5938,0.0000
C01391=-28.763,35.614,12.332,148.7645,24.5871,0.0000
C01392=-27.143,37.028,12.387,149.4044,25.1888,0.0000
C01393=-26.243,38.108,12.523,149.8901,25.5837,0.0000
C01394=-25.839,39.052,12.705,150.2497,25.8397,0.0000
C01395=-25.668,39.997,12.887,150.5670,26.0379,0.0000
C01396=-25.514,40.979,13.022,150.9073,26.2307,0.0000
C01397=-25.133,42.005,13.088,151.3503,26.4769,0.0000
C01398=-24.255,43.149,13.123,152.0216,26.8513,0.0000
C01399=-22.974,44.253,13.151,152.8610,27.2983,0.0000
C01400=-21.465,45.136,13.179,153.7450,27.7420,0.0000
C01401=-19.915,45.860,13.197,154.6177,28.1428,0.0000
C01402=-18.347,46.510,13.197,142.9785,-3.7987,0.0000
C01403=-16.738,47.094,13.179,142.6395,-2.9983,0.0000
C01404=-15.047,47.537,13.151,142.3125,-2.1588,0.0000
C01405=-13.360,47.661,13.123,142.0105,-1.3420,0.0000
C01406=-11.930,47.474,13.088,141.7742,-0.6754,0.0000
C01407=-10.935,47.018,13.022,141.6149,-0.2364,0.0000
C01408=-10.132,46.432,12.887,141.4934,0.1039,0.0000
C01409=-9.343,45.885,12.705,141.3902,0.4356,0.0000
C01410=-8.390,45.503,12.523,141.2910,0.8365,0.0000
C01411=-6.990,45.375,12.387,141.1845,1.4171,0.0000
C01412=-4.844,45.521,12.332,141.0883,2.2477,0.0000
C01413=-2.510,45.702,12.329,141.0371,2.2781,0.0000
C01414=0.000,45.772,12.331,140.9966,0.0004,0.0000
C01415=0.000,44.574,14.176,140.8479,0.0003,0.0000
C01416=2.400,44.508,14.174,140.8887,-2.2694,0.0000
C01417=4.660,44.338,14.177,140.9369,-2.2137,0.0000
C01418=6.764,44.232,14.253,141.0278,-1.3642,0.0000
C01419=8.113,44.459,14.440,141.1266,-0.7874,0.0000
C01420=9.024,44.998,14.693,141.2170,-0.3974,0.0000
C01421=9.783,45.750,14.949,141.3117,-0.0755,0.0000
C01422=10.558,46.569,15.143,141.4249,0.2538,0.0000
C01423=11.519,47.250,15.238,141.5763,0.6800,0.0000
C01424=12.971,47.615,15.288,141.8148,1.3698,0.0000
C01425=14.738,47.593,15.328,142.1339,2.2469,0.0000
C01426=16.543,47.159,15.369,142.4925,3.1675,0.0000
C01427=18.280,46.536,15.396,142.8740,4.0537,0.0000
C01428=19.980,45.832,15.396,154.7123,-28.4054,0.0000
C01429=21.649,45.044,15.369,153.7382,-27.9660,0.0000
C01430=23.232,44.075,15.328,152.7673,-27.4790,0.0000
C01431=24.496,42.841,15.288,151.8696,-26.9952,0.0000
C01432=25.266,41.555,15.238,151.1799,-26.6031,0.0000
C01433=25.464,40.395,15.143,150.7527,-26.3617,0.0000
C01434=25.432,39.268,14.949,150.4270,-26.1721,0.0000
C01435=25.438,38.199,14.693,150.1237,-25.9761,0.0000
C01436=25.701,37.174,14.440,149.7790,-25.7231,0.0000
C01437=26.493,36.060,14.253,149.3026,-25.3261,0.0000
C01438=28.056,34.647,14.177,148.6545,-24.7056,0.0000
C01439=29.775,33.169,14.174,148.5752,-24.6903,0.0000
C01440=31.519,31.519,14.176,150.0703,-26.5167,0.0000
C01441=33.169,29.775,14.174,151.6855,-28.2755,0.0000
C01442=34.647,28.056,14.177,151.6888,-28.2017,0.0000
C01443=36.060,26.493,14.253,151.1723,-27.4795,0.0000
C01444=37.174,25.701,14.440,150.8583,-26.9653,0.0000
C01445=38.199,25.438,14.693,150.6685,-26.6027,0.0000
C01446=39.268,25.432,14.949,150.5304,-26.2908,0.0000
C01447=40.395,25.464,15.143,150.4042,-25.9615,0.0000
C01448=41.555,25.266,15.238,150.2461,-25.5324,0.0000
C01449=42.841,24.496,15.288,149.9868,-24.8413,0.0000
C01450=44.075,23.232,15.328,149.6749,-23.9523,0.0000
C01451=45.044,21.649,15.369,149.3720,-23.0045,0.0000
C01452=45.832,19.980,15.396,149.1149,-22.0697,0.0000
C01453=46.536,18.280,15.396,-174.9206,-37.0176,0.0000
C01454=47.159,16.543,15.369,-176.0094,-37.4404,0.0000
C01455=47.593,14.738,15.328,-177.1547,-37.8318,0.0000
C01456=47.615,12.971,15.288,-178.2575,-38.1724,0.0000
C01457=47.250,11.519,15.238,-179.1321,-38.4205,0.0000
C01458=46.569,10.558,15.143,-179.6754,-38.5746,0.0000
C01459=45.750,9.783,14.949,179.9032,-38.6883,0.0000
C01460=44.998,9.024,14.693,179.4902,-38.7819,0.0000
C01461=44.459,8.113,14.440,178.9887,-38.8691,0.0000
C01462=44.232,6.764,14.253,178.2455,-38.9591,0.0000
C01463=44.338,4.660,14.177,177.1499,-39.0284,0.0000
C01464=44.508,2.400,14.174,177.0763,-39.0748,0.0000
C01465=44.574,0.000,14.176,-179.9996,-39.1521,0.0000
C01466=44.508,-2.400,14.174,-177.0765,-39.0749,0.0000
C01467=44.338,-4.660,14.177,-177.1504,-39.0284,0.0000
C01468=44.232,-6.764,14.253,-178.2462,-38.9590,0.0000
C01469=44.459,-8.113,14.440,-178.9893,-38.8690,0.0000
C01470=44.998,-9.024,14.693,-179.4907,-38.7818,0.0000
C01471=45.750,-9.783,14.949,-179.9037,-38.6882,0.0000
C01472=46.569,-10.558,15.143,179.6749,-38.5746,0.0000
C01473=47.250,-11.519,15.238,179.1317,-38.4205,0.0000
C01474=47.615,-12.971,15.288,178.2572,-38.1723,0.0000
C01475=47.593,-14.738,15.328,177.1546,-37.8318,0.0000
C01476=47.159,-16.543,15.369,176.0094,-37.4403,0.0000
C01477=46.536,-18.280,15.396,174.9207,-37.0175,0.0000
C01478=45.832,-19.980,15.396,-149.1148,-22.0697,0.0000
C01479=45.044,-21.649,15.369,-149.3720,-23.0045,0.0000
C01480=44.075,-23.232,15.328,-149.6749,-23.9524,0.0000
C01481=42.841,-24.496,15.288,-149.9869,-24.8415,0.0000
C01482=41.555,-25.266,15.238,-150.2462,-25.5326,0.0000
C01483=40.395,-25.464,15.143,-150.4044,-25.9619,0.0000
C01484=39.268,-25.432,14.949,-150.5306,-26.2911,0.0000
C01485=38.199,-25.438,14.693,-150.6688,-26.6030,0.0000
C01486=37.174,-25.701,14.440,-150.8586,-26.9657,0.0000
C01487=36.060,-26.493,14.253,-151.1726,-27.4800,0.0000
C01488=34.647,-28.056,14.177,-151.6890,-28.2020,0.0000
C01489=33.169,-29.775,14.174,-151.6856,-28.2756,0.0000
C01490=31.519,-31.519,14.176,-150.0699,-26.5162,0.0000
C01491=29.775,-33.169,14.174,-148.5753,-24.6905,0.0000
C01492=28.056,-34.647,14.177,-148.6548,-24.7059,0.0000
C01493=26.493,-36.060,14.253,-149.3030,-25.3265,0.0000
C01494=25.701,-37.174,14.440,-149.7794,-25.7235,0.0000
C01495=25.438,-38.199,14.693,-150.1240,-25.9765,0.0000
C01496=25.432,-39.268,14.949,-150.4273,-26.1723,0.0000
C01497=25.464,-40.395,15.143,-150.7529,-26.3620,0.0000
C01498=25.266,-41.555,15.238,-151.1802,-26.6033,0.0000
C01499=24.496,-42.841,15.288,-151.8698,-26.9954,0.0000
C01500=23.232,-44.075,15.328,-152.7674,-27.4791,0.0000
C01501=21.649,-45.044,15.369,-153.7383,-27.9659,0.0000
C01502=19.980,-45.832,15.396,-154.7123,-28.4053,0.0000
C01503=18.280,-46.536,15.396,-142.8740,4.0537,0.0000
C01504=16.543,-47.159,15.369,-142.4925,3.1675,0.0000
C01505=14.738,-47.593,15.328,-142.1339,2.2469,0.0000
C01506=12.971,-47.615,15.288,-141.8148,1.3698,0.0000
C01507=11.519,-47.250,15.238,-141.5763,0.6800,0.0000
C01508=10.558,-46.569,15.143,-141.4249,0.2538,0.0000
C01509=9.783,-45.750,14.949,-141.3117,-0.0755,0.0000
C01510=9.024,-44.998,14.693,-141.2170,-0.3974,0.0000
C01511=8.113,-44.459,14.440,-141.1266,-0.7874,0.0000
C01512=6.764,-44.232,14.253,-141.0278,-1.3642,0.0000
C01513=4.660,-44.338,14.177,-140.9369,-2.2137,0.0000
C01514=2.400,-44.508,14.174,-140.8887,-2.2694,0.0000
C01515=0.000,-44.574,14.176,-140.8479,0.0003,0.0000
C01516=0.000,-44.574,14.176,-140.8479,0.0003,0.0000
C01517=-2.400,-44.508,14.174,-140.8886,2.2692,0.0000
C01518=-4.660,-44.338,14.177,-140.9369,2.2133,0.0000
C01519=-6.764,-44.232,14.253,-141.0279,1.3637,0.0000
C01520=-8.113,-44.459,14.440,-141.1266,0.7869,0.0000
C01521=-9.024,-44.998,14.693,-141.2171,0.3970,0.0000
C01522=-9.783,-45.750,14.949,-141.3117,0.0751,0.0000
C01523=-10.558,-46.569,15.143,-141.4250,-0.2541,0.0000
C01524=-11.519,-47.250,15.238,-141.5763,-0.6802,0.0000
C01525=-12.971,-47.615,15.288,-141.8148,-1.3700,0.0000
C01526=-14.738,-47.593,15.328,-142.1340,-2.2470,0.0000
C01527=-16.543,-47.159,15.369,-142.4925,-3.1675,0.0000
C01528=-18.280,-46.536,15.396,-142.8740,-4.0536,0.0000
C01529=-19.980,-45.832,15.396,-154.7123,28.4054,0.0000
C01530=-21.649,-45.044,15.369,-153.7382,27.9660,0.0000
C01531=-23.232,-44.075,15.328,-152.7673,27.4790,0.0000
C01532=-24.496,-42.841,15.288,-151.8696,26.9952,0.0000
C01533=-25.266,-41.555,15.238,-151.1799,26.6031,0.0000
C01534=-25.464,-40.395,15.143,-150.7527,26.3617,0.0000
C01535=-25.432,-39.268,14.949,-150.4270,26.1721,0.0000
C01536=-25.438,-38.199,14.693,-150.1237,25.9761,0.0000
C01537=-25.701,-37.174,14.440,-149.7790,25.7231,0.0000
C01538=-26.493,-36.060,14.253,-149.3026,25.3261,0.0000
C01539=-28.056,-34.647,14.177,-148.6545,24.7056,0.0000
C01540=-29.775,-33.169,14.174,-148.5752,24.6903,0.0000
C01541=-31.519,-31.519,14.176,-150.0703,26.5167,0.0000
C01542=-33.169,-29.775,14.174,-151.6855,28.2755,0.0000
C01543=-34.647,-28.056,14.177,-151.6888,28.2017,0.0000
C01544=-36.060,-26.493,14.253,-151.1723,27.4795,0.0000
C01545=-37.174,-25.701,14.440,-150.8583,26.9653,0.0000
C01546=-38.199,-25.438,14.693,-150.6685,26.6027,0.0000
C01547=-39.268,-25.432,14.949,-150.5304,26.2908,0.0000
C01548=-40.395,-25.464,15.143,-150.4042,25.9615,0.0000
C01549=-41.555,-25.266,15.238,-150.2461,25.5324,0.0000
C01550=-42.841,-24.496,15.288,-149.9868,24.8413,0.0000
C01551=-44.075,-23.232,15.328,-149.6749,23.9523,0.0000
C01552=-45.044,-21.649,15.369,-149.3720,23.0045,0.0000
C01553=-45.832,-19.980,15.396,-149.1149,22.0697,0.0000
C01554=-46.536,-18.280,15.396,174.9206,37.0176,0.0000
C01555=-47.159,-16.543,15.369,176.0094,37.4404,0.0000
C01556=-47.593,-14.738,15.328,177.1547,37.8318,0.0000
C01557=-47.615,-12.971,15.288,178.2575,38.1724,0.0000
C01558=-47.250,-11.519,15.238,179.1321,38.4205,0.0000
C01559=-46.569,-10.558,15.143,179.6754,38.5746,0.0000
C01560=-45.750,-9.783,14.949,-179.9032,38.6883,0.0000
C01561=-44.998,-9.024,14.693,-179.4902,38.7819,0.0000
C01562=-44.459,-8.113,14.440,-178.9887,38.8691,0.0000
C01563=-44.232,-6.764,14.253,-178.2455,38.9591,0.0000
C01564=-44.338,-4.660,14.177,-177.1499,39.0284,0.0000
C01565=-44.508,-2.400,14.174,-177.0763,39.0748,0.0000
C01566=-44.574,0.000,14.176,179.9996,39.1521,0.0000
C01567=-44.508,2.400,14.174,177.0765,39.0749,0.0000
C01568=-44.338,4.660,14.177,177.1504,39.0284,0.0000
C01569=-44.232,6.764,14.253,178.2462,38.9590,0.0000
C01570=-44.459,8.113,14.440,178.9893,38.8690,0.0000
C01571=-44.998,9.024,14.693,179.4907,38.7818,0.0000
C01572=-45.750,9.783,14.949,179.9037,38.6882,0.0000
C01573=-46.569,10.558,15.143,-179.6749,38.5746,0.0000
C01574=-47.250,11.519,15.238,-179.1317,38.4205,0.0000
C01575=-47.615,12.971,15.288,-178.2572,38.1723,0.0000
C01576=-47.593,14.738,15.328,-177.1546,37.8318,0.0000
C01577=-47.159,16.543,15.369,-176.0094,37.4403,0.0000
C01578=-46.536,18.280,15.396,-174.9207,37.0175,0.0000
C01579=-45.832,19.980,15.396,149.1148,22.0697,0.0000
C01580=-45.044,21.649,15.369,149.3720,23.0045,0.0000
C01581=-44.075,23.232,15.328,149.6749,23.9524,0.0000
C01582=-42.841,24.496,15.288,149.9869,24.8415,0.0000
C01583=-41.555,25.266,15.238,150.2462,25.5326,0.0000
C01584=-40.395,25.464,15.143,150.4044,25.9619,0.0000
C01585=-39.268,25.432,14.949,150.5306,26.2911,0.0000
C01586=-38.199,25.438,14.693,150.6688,26.6030,0.0000
C01587=-37.174,25.701,14.440,150.8586,26.9657,0.0000
C01588=-36.060,26.493,14.253,151.1726,27.4800,0.0000
C01589=-34.647,28.056,14.177,151.6890,28.2020,0.0000
C01590=-33.169,29.775,14.174,151.6856,28.2756,0.0000
C01591=-31.519,31.519,14.176,150.0699,26.5162,0.0000
C01592=-29.775,33.169,14.174,148.5753,24.6905,0.0000
C01593=-28.056,34.647,14.177,148.6548,24.7059,0.0000
C01594=-26.493,36.060,14.253,149.3030,25.3265,0.0000
C01595=-25.701,37.174,14.440,149.7794,25.7235,0.0000
C01596=-25.438,38.199,14.693,150.1240,25.9765,0.0000
C01597=-25.432,39.268,14.949,150.4273,26.1723,0.0000
C01598=-25.464,40.395,15.143,150.7529,26.3620,0.0000
C01599=-25.266,41.555,15.238,151.1802,26.6033,0.0000
C01600=-24.496,42.841,15.288,151.8698,26.9954,0.0000
C01601=-23.232,44.075,15.328,152.7674,27.4791,0.0000
C01602=-21.649,45.044,15.369,153.7383,27.9659,0.0000
C01603=-19.980,45.832,15.396,154.7123,28.4053,0.0000
C01604=-18.280,46.536,15.396,142.8740,-4.0536,0.0000
C01605=-16.543,47.159,15.369,142.4925,-3.1675,0.0000
C01606=-14.738,47.593,15.328,142.1340,-2.2470,0.0000
C01607=-12.971,47.615,15.288,141.8148,-1.3700,0.0000
C01608=-11.519,47.250,15.238,141.5763,-0.6802,0.0000
C01609=-10.558,46.569,15.143,141.4250,-0.2541,0.0000
C01610=-9.783,45.750,14.949,141.3117,0.0751,0.0000
C01611=-9.024,44.998,14.693,141.2171,0.3970,0.0000
C01612=-8.113,44.459,14.440,141.1266,0.7869,0.0000
C01613=-6.764,44.232,14.253,141.0279,1.3637,0.0000
C01614=-4.660,44.338,14.177,140.9369,2.2133,0.0000
C01615=-2.400,44.508,14.174,140.8886,2.2692,0.0000
C01616=0.000,44.574,14.176,140.8479,0.0003,0.0000
C01617=0.000,43.311,15.978,140.7557,0.0002,0.0000
C01618=2.285,43.249,15.975,140.7966,-2.2547,0.0000
C01619=4.466,43.090,15.979,140.8421,-2.1834,0.0000
C01620=6.526,43.024,16.076,140.9276,-1.3211,0.0000
C01621=7.820,43.354,16.319,141.0177,-0.7532,0.0000
C01622=8.685,44.055,16.652,141.0976,-0.3771,0.0000
C01623=9.411,45.022,16.991,141.1807,-0.0683,0.0000
C01624=10.154,46.088,17.251,141.2815,0.2470,0.0000
C01625=11.076,47.009,17.379,141.4201,0.6569,0.0000
C01626=12.553,47.564,17.447,141.6566,1.3704,0.0000
C01627=14.406,47.654,17.502,141.9915,2.3126,0.0000
C01628=16.332,47.228,17.558,142.3839,3.3218,0.0000
C01629=18.209,46.563,17.595,142.8130,4.3017,0.0000
C01630=20.050,45.800,17.595,154.8402,-28.6347,0.0000
C01631=21.847,44.944,17.558,153.7544,-28.1540,0.0000
C01632=23.510,43.883,17.502,152.6891,-27.6196,0.0000
C01633=24.756,42.510,17.447,151.7313,-27.0942,0.0000
C01634=25.408,41.072,17.379,151.0267,-26.6817,0.0000
C01635=25.409,39.769,17.251,150.6219,-26.4448,0.0000
C01636=25.181,38.490,16.991,150.3168,-26.2582,0.0000
C01637=25.011,37.293,16.652,150.0326,-26.0654,0.0000
C01638=25.126,36.186,16.319,149.7065,-25.8166,0.0000
C01639=25.808,35.038,16.076,149.2436,-25.4213,0.0000
C01640=27.311,33.628,15.979,148.5916,-24.7870,0.0000
C01641=28.966,32.197,15.975,148.5042,-24.7576,0.0000
C01642=30.625,30.625,15.978,149.9888,-26.5730,0.0000
C01643=32.197,28.966,15.975,151.5933,-28.3213,0.0000
C01644=33.628,27.311,15.979,151.5832,-28.2370,0.0000
C01645=35.038,25.808,16.076,151.0536,-27.5077,0.0000
C01646=36.186,25.126,16.319,150.7386,-27.0056,0.0000
C01647=37.293,25.011,16.652,150.5493,-26.6602,0.0000
C01648=38.490,25.181,16.991,150.4102,-26.3657,0.0000
C01649=39.769,25.409,17.251,150.2829,-26.0550,0.0000
C01650=41.072,25.408,17.379,150.1250,-25.6464,0.0000
C01651=42.510,24.756,17.447,149.8486,-24.9375,0.0000
C01652=43.883,23.510,17.502,149.5076,-23.9871,0.0000
C01653=44.944,21.847,17.558,149.1765,-22.9481,0.0000
C01654=45.800,20.050,17.595,148.9002,-21.9097,0.0000
C01655=46.563,18.209,17.595,-174.6062,-37.0647,0.0000
C01656=47.228,16.332,17.558,-175.8092,-37.5420,0.0000
C01657=47.654,14.406,17.502,-177.0659,-37.9720,0.0000
C01658=47.564,12.553,17.447,-178.2529,-38.3304,0.0000
C01659=47.009,11.076,17.379,-179.1598,-38.5769,0.0000
C01660=46.088,10.154,17.251,-179.6835,-38.7180,0.0000
C01661=45.022,9.411,16.991,179.9123,-38.8192,0.0000
C01662=44.055,8.685,16.652,179.5155,-38.9014,0.0000
C01663=43.354,7.820,16.319,179.0311,-38.9782,0.0000
C01664=43.024,6.526,16.076,178.2986,-39.0601,0.0000
C01665=43.090,4.466,15.979,177.1852,-39.1241,0.0000
C01666=43.249,2.285,15.975,177.0914,-39.1673,0.0000
C01667=43.311,0.000,15.978,-179.9998,-39.2443,0.0000
C01668=43.249,-2.285,15.975,-177.0916,-39.1673,0.0000
C01669=43.090,-4.466,15.979,-177.1857,-39.1240,0.0000
C01670=43.024,-6.526,16.076,-178.2992,-39.0600,0.0000
C01671=43.354,-7.820,16.319,-179.0317,-38.9782,0.0000
C01672=44.055,-8.685,16.652,-179.5161,-38.9013,0.0000
C01673=45.022,-9.411,16.991,-179.9128,-38.8192,0.0000
C01674=46.088,-10.154,17.251,179.6830,-38.7180,0.0000
C01675=47.009,-11.076,17.379,179.1594,-38.5769,0.0000
C01676=47.564,-12.553,17.447,178.2526,-38.3303,0.0000
C01677=47.654,-14.406,17.502,177.0657,-37.9720,0.0000
C01678=47.228,-16.332,17.558,175.8092,-37.5420,0.0000
C01679=46.563,-18.209,17.595,174.6062,-37.0646,0.0000
C01680=45.800,-20.050,17.595,-148.9001,-21.9097,0.0000
C01681=44.944,-21.847,17.558,-149.1765,-22.9481,0.0000
C01682=43.883,-23.510,17.502,-149.5077,-23.9872,0.0000
C01683=42.510,-24.756,17.447,-149.8487,-24.9377,0.0000
C01684=41.072,-25.408,17.379,-150.1252,-25.6467,0.0000
C01685=39.769,-25.409,17.251,-150.2831,-26.0553,0.0000
C01686=38.490,-25.181,16.991,-150.4105,-26.3660,0.0000
C01687=37.293,-25.011,16.652,-150.5495,-26.6605,0.0000
C01688=36.186,-25.126,16.319,-150.7389,-27.0060,0.0000
C01689=35.038,-25.808,16.076,-151.0538,-27.5081,0.0000
C01690=33.628,-27.311,15.979,-151.5835,-28.2373,0.0000
C01691=32.197,-28.966,15.975,-151.5935,-28.3214,0.0000
C01692=30.625,-30.625,15.978,-149.9886,-26.5727,0.0000
C01693=28.966,-32.197,15.975,-148.5043,-24.7578,0.0000
C01694=27.311,-33.628,15.979,-148.5918,-24.7873,0.0000
C01695=25.808,-35.038,16.076,-149.2440,-25.4216,0.0000
C01696=25.126,-36.186,16.319,-149.7069,-25.8170,0.0000
C01697=25.011,-37.293,16.652,-150.0330,-26.0657,0.0000
C01698=25.181,-38.490,16.991,-150.3171,-26.2585,0.0000
C01699=25.409,-39.769,17.251,-150.6222,-26.4450,0.0000
C01700=25.408,-41.072,17.379,-151.0270,-26.6819,0.0000
C01701=24.756,-42.510,17.447,-151.7315,-27.0944,0.0000
C01702=23.510,-43.883,17.502,-152.6893,-27.6197,0.0000
C01703=21.847,-44.944,17.558,-153.7544,-28.1540,0.0000
C01704=20.050,-45.800,17.595,-154.8402,-28.6347,0.0000
C01705=18.209,-46.563,17.595,-142.8130,4.3017,0.0000
C01706=16.332,-47.228,17.558,-142.3839,3.3218,0.0000
C01707=14.406,-47.654,17.502,-141.9915,2.3126,0.0000
C01708=12.553,-47.564,17.447,-141.6566,1.3704,0.0000
C01709=11.076,-47.009,17.379,-141.4201,0.6569,0.0000
C01710=10.154,-46.088,17.251,-141.2815,0.2470,0.0000
C01711=9.411,-45.022,16.991,-141.1807,-0.0683,0.0000
C01712=8.685,-44.055,16.652,-141.0976,-0.3771,0.0000
C01713=7.820,-43.354,16.319,-141.0177,-0.7532,0.0000
C01714=6.526,-43.024,16.076,-140.9276,-1.3211,0.0000
C01715=4.466,-43.090,15.979,-140.8421,-2.1834,0.0000
C01716=2.285,-43.249,15.975,-140.7966,-2.2547,0.0000
C01717=0.000,-43.311,15.978,-140.7557,0.0002,0.0000
C01718=0.000,-43.311,15.978,-140.7557,0.0002,0.0000
C01719=-2.285,-43.249,15.975,-140.7965,2.2545,0.0000
C01720=-4.466,-43.090,15.979,-140.8421,2.1830,0.0000
C01721=-6.526,-43.024,16.076,-140.9276,1.3206,0.0000
C01722=-7.820,-43.354,16.319,-141.0178,0.7528,0.0000
C01723=-8.685,-44.055,16.652,-141.0977,0.3766,0.0000
C01724=-9.411,-45.022,16.991,-141.1808,0.0679,0.0000
C01725=-10.154,-46.088,17.251,-141.2816,-0.2473,0.0000
C01726=-11.076,-47.009,17.379,-141.4201,-0.6572,0.0000
C01727=-12.553,-47.564,17.447,-141.6567,-1.3706,0.0000
C01728=-14.406,-47.654,17.502,-141.9915,-2.3128,0.0000
C01729=-16.332,-47.228,17.558,-142.3839,-3.3218,0.0000
C01730=-18.209,-46.563,17.595,-142.8130,-4.3017,0.0000
C01731=-20.050,-45.800,17.595,-154.8402,28.6347,0.0000
C01732=-21.847,-44.944,17.558,-153.7544,28.1540,0.0000
C01733=-23.510,-43.883,17.502,-152.6891,27.6196,0.0000
C01734=-24.756,-42.510,17.447,-151.7313,27.0942,0.0000
C01735=-25.408,-41.072,17.379,-151.0267,26.6817,0.0000
C01736=-25.409,-39.769,17.251,-150.6219,26.4448,0.0000
C01737=-25.181,-38.490,16.991,-150.3168,26.2582,0.0000
C01738=-25.011,-37.293,16.652,-150.0326,26.0654,0.0000
C01739=-25.126,-36.186,16.319,-149.7065,25.8166,0.0000
C01740=-25.808,-35.038,16.076,-149.2436,25.4213,0.0000
C01741=-27.311,-33.628,15.979,-148.5916,24.7870,0.0000
C01742=-28.966,-32.197,15.975,-148.5042,24.7576,0.0000
C01743=-30.625,-30.625,15.978,-149.9888,26.5730,0.0000
C01744=-32.197,-28.966,15.975,-151.5933,28.3213,0.0000
C01745=-33.628,-27.311,15.979,-151.5832,28.2370,0.0000
C01746=-35.038,-25.808,16.076,-151.0536,27.5077,0.0000
C01747=-36.186,-25.126,16.319,-150.7386,27.0056,0.0000
C01748=-37.293,-25.011,16.652,-150.5493,26.6602,0.0000
C01749=-38.490,-25.181,16.991,-150.4102,26.3657,0.0000
C01750=-39.769,-25.409,17.251,-150.2829,26.0550,0.0000
C01751=-41.072,-25.408,17.379,-150.1250,25.6464,0.0000
C01752=-42.510,-24.756,17.447,-149.8486,24.9375,0.0000
C01753=-43.883,-23.510,17.502,-149.5076,23.9871,0.0000
C01754=-44.944,-21.847,17.558,-149.1765,22.9481,0.0000
C01755=-45.800,-20.050,17.595,-148.9002,21.9097,0.0000
C01756=-46.563,-18.209,17.595,174.6062,37.0647,0.0000
C01757=-47.228,-16.332,17.558,175.8092,37.5420,0.0000
C01758=-47.654,-14.406,17.502,177.0659,37.9720,0.0000
C01759=-47.564,-12.553,17.447,178.2529,38.3304,0.0000
C01760=-47.009,-11.076,17.379,179.1598,38.5769,0.0000
C01761=-46.088,-10.154,17.251,179.6835,38.7180,0.0000
C01762=-45.022,-9.411,16.991,-179.9123,38.8192,0.0000
C01763=-44.055,-8.685,16.652,-179.5155,38.9014,0.0000
C01764=-43.354,-7.820,16.319,-179.0311,38.9782,0.0000
C01765=-43.024,-6.526,16.076,-178.2986,39.0601,0.0000
C01766=-43.090,-4.466,15.979,-177.1852,39.1241,0.0000
C01767=-43.249,-2.285,15.975,-177.0914,39.1673,0.0000
C01768=-43.311,0.000,15.978,179.9998,39.2443,0.0000
C01769=-43.249,2.285,15.975,177.0916,39.1673,0.0000
C01770=-43.090,4.466,15.979,177.1857,39.1240,0.0000
C01771=-43.024,6.526,16.076,178.2992,39.0600,0.0000
C01772=-43.354,7.820,16.319,179.0317,38.9782,0.0000
C01773=-44.055,8.685,16.652,179.5161,38.9013,0.0000
C01774=-45.022,9.411,16.991,179.9128,38.8192,0.0000
C01775=-46.088,10.154,17.251,-179.6830,38.7180,0.0000
C01776=-47.009,11.076,17.379,-179.1594,38.5769,0.0000
C01777=-47.564,12.553,17.447,-178.2526,38.3303,0.0000
C01778=-47.654,14.406,17.502,-177.0657,37.9720,0.0000
C01779=-47.228,16.332,17.558,-175.8092,37.5420,0.0000
C01780=-46.563,18.209,17.595,-174.6062,37.0646,0.0000
C01781=-45.800,20.050,17.595,148.9001,21.9097,0.0000
C01782=-44.944,21.847,17.558,149.1765,22.9481,0.0000
C01783=-43.883,23.510,17.502,149.5077,23.9872,0.0000
C01784=-42.510,24.756,17.447,149.8487,24.9377,0.0000
C01785=-41.072,25.408,17.379,150.1252,25.6467,0.0000
C01786=-39.769,25.409,17.251,150.2831,26.0553,0.0000
C01787=-38.490,25.181,16.991,150.4105,26.3660,0.0000
C01788=-37.293,25.011,16.652,150.5495,26.6605,0.0000
C01789=-36.186,25.126,16.319,150.7389,27.0060,0.0000
C01790=-35.038,25.808,16.076,151.0538,27.5081,0.0000
C01791=-33.628,27.311,15.979,151.5835,28.2373,0.0000
C01792=-32.197,28.966,15.975,151.5935,28.3214,0.0000
C01793=-30.625,30.625,15.978,149.9886,26.5727,0.0000
C01794=-28.966,32.197,15.975,148.5043,24.7578,0.0000
C01795=-27.311,33.628,15.979,148.5918,24.7873,0.0000
C01796=-25.808,35.038,16.076,149.2440,25.4216,0.0000
C01797=-25.126,36.186,16.319,149.7069,25.8170,0.0000
C01798=-25.011,37.293,16.652,150.0330,26.0657,0.0000
C01799=-25.181,38.490,16.991,150.3171,26.2585,0.0000
C01800=-25.409,39.769,17.251,150.6222,26.4450,0.0000
C01801=-25.408,41.072,17.379,151.0270,26.6819,0.0000
C01802=-24.756,42.510,17.447,151.7315,27.0944,0.0000
C01803=-23.510,43.883,17.502,152.6893,27.6197,0.0000
C01804=-21.847,44.944,17.558,153.7544,28.1540,0.0000
C01805=-20.050,45.800,17.595,154.8402,28.6347,0.0000
C01806=-18.209,46.563,17.595,142.8130,-4.3017,0.0000
C01807=-16.332,47.228,17.558,142.3839,-3.3218,0.0000
C01808=-14.406,47.654,17.502,141.9915,-2.3128,0.0000
C01809=-12.553,47.564,17.447,141.6567,-1.3706,0.0000
C01810=-11.076,47.009,17.379,141.4201,-0.6572,0.0000
C01811=-10.154,46.088,17.251,141.2816,-0.2473,0.0000
C01812=-9.411,45.022,16.991,141.1808,0.0679,0.0000
C01813=-8.685,44.055,16.652,141.0977,0.3766,0.0000
C01814=-7.820,43.354,16.319,141.0178,0.7528,0.0000
C01815=-6.526,43.024,16.076,140.9276,1.3206,0.0000
C01816=-4.466,43.090,15.979,140.8421,2.1830,0.0000
C01817=-2.285,43.249,15.975,140.7965,2.2545,0.0000
C01818=0.000,43.311,15.978,140.7557,0.0002,0.0000
C01819=0.000,41.999,17.743,140.7155,0.0000,0.0000
C01820=2.165,41.942,17.740,140.7562,-2.2346,0.0000
C01821=4.264,41.794,17.745,140.7991,-2.1569,0.0000
C01822=6.279,41.769,17.866,140.8792,-1.2875,0.0000
C01823=7.515,42.203,18.169,140.9602,-0.7332,0.0000
C01824=8.331,43.070,18.587,141.0282,-0.3734,0.0000
C01825=9.020,44.258,19.017,141.0971,-0.0802,0.0000
C01826=9.729,45.582,19.349,141.1816,0.2186,0.0000
C01827=10.611,46.755,19.514,141.3027,0.6094,0.0000
C01828=12.113,47.511,19.602,141.5332,1.3471,0.0000
C01829=14.056,47.717,19.673,141.8819,2.3590,0.0000
C01830=16.110,47.302,19.746,142.3101,3.4636,0.0000
C01831=18.133,46.592,19.794,142.7916,4.5442,0.0000
C01832=20.124,45.768,19.794,154.9993,-28.8342,0.0000
C01833=22.056,44.839,19.746,153.7921,-28.3103,0.0000
C01834=23.802,43.680,19.673,152.6258,-27.7245,0.0000
C01835=25.030,42.161,19.602,151.6064,-27.1528,0.0000
C01836=25.558,40.564,19.514,150.8906,-26.7169,0.0000
C01837=25.352,39.110,19.349,150.5144,-26.4840,0.0000
C01838=24.917,37.674,19.017,150.2350,-26.3002,0.0000
C01839=24.565,36.346,18.587,149.9740,-26.1108,0.0000
C01840=24.528,35.156,18.169,149.6695,-25.8676,0.0000
C01841=25.096,33.975,17.866,149.2236,-25.4773,0.0000
C01842=26.538,32.569,17.745,148.5715,-24.8340,0.0000
C01843=28.126,31.188,17.740,148.4821,-24.7980,0.0000
C01844=29.698,29.698,17.743,149.9532,-26.5976,0.0000
C01845=31.188,28.126,17.740,151.5431,-28.3307,0.0000
C01846=32.569,26.538,17.745,151.5264,-28.2430,0.0000
C01847=33.975,25.096,17.866,150.9873,-27.5113,0.0000
C01848=35.156,24.528,18.169,150.6739,-27.0253,0.0000
C01849=36.346,24.565,18.587,150.4855,-26.7000,0.0000
C01850=37.674,24.917,19.017,150.3448,-26.4264,0.0000
C01851=39.110,25.352,19.349,150.2144,-26.1388,0.0000
C01852=40.564,25.558,19.514,150.0544,-25.7559,0.0000
C01853=42.161,25.030,19.602,149.7565,-25.0315,0.0000
C01854=43.680,23.802,19.673,149.3816,-24.0171,0.0000
C01855=44.839,22.056,19.746,149.0194,-22.8803,0.0000
C01856=45.768,20.124,19.794,148.7235,-21.7299,0.0000
C01857=46.592,18.133,19.794,-174.3013,-37.0717,0.0000
C01858=47.302,16.110,19.746,-175.6262,-37.6091,0.0000
C01859=47.717,14.056,19.673,-177.0026,-38.0801,0.0000
C01860=47.511,12.113,19.602,-178.2797,-38.4543,0.0000
C01861=46.755,10.611,19.514,-179.2192,-38.6947,0.0000
C01862=45.582,9.729,19.349,-179.7194,-38.8181,0.0000
C01863=44.258,9.020,19.017,179.8969,-38.9028,0.0000
C01864=43.070,8.331,18.587,179.5197,-38.9709,0.0000
C01865=42.203,7.515,18.169,179.0561,-39.0360,0.0000
C01866=41.769,6.279,17.866,178.3407,-39.1090,0.0000
C01867=41.794,4.264,17.745,177.2175,-39.1678,0.0000
C01868=41.942,2.165,17.740,177.1156,-39.2083,0.0000
C01869=41.999,0.000,17.743,-179.9999,-39.2845,0.0000
C01870=41.942,-2.165,17.740,-177.1159,-39.2083,0.0000
C01871=41.794,-4.265,17.745,-177.2181,-39.1678,0.0000
C01872=41.769,-6.279,17.866,-178.3413,-39.1090,0.0000
C01873=42.203,-7.515,18.169,-179.0567,-39.0359,0.0000
C01874=43.070,-8.331,18.587,-179.5203,-38.9708,0.0000
C01875=44.258,-9.020,19.017,-179.8974,-38.9028,0.0000
C01876=45.582,-9.729,19.349,179.7189,-38.8180,0.0000
C01877=46.755,-10.611,19.514,179.2188,-38.6946,0.0000
C01878=47.511,-12.113,19.602,178.2794,-38.4542,0.0000
C01879=47.717,-14.056,19.673,177.0025,-38.0800,0.0000
C01880=47.302,-16.110,19.746,175.6262,-37.6091,0.0000
C01881=46.592,-18.133,19.794,174.3014,-37.0717,0.0000
